LIN {X 0,Y 428.465,Z 323.366,A -85,B 0,C 180,E1 -10193.855,E2 -10193.855} C_VEL
LIN {X 0,Y 430.583,Z 198.986,A -85,B 0,C 180,E1 -10195.968,E2 -10195.968} C_VEL
LIN {X 0,Y 425.08,Z 170.607,A -85,B 0,C 180,E1 -10196.85,E2 -10196.85} C_VEL
LIN {X 0,Y 424.032,Z 165.531,A -85,B 0,C 180,E1 -10197.037,E2 -10197.037} C_VEL
LIN {X 0,Y 424.428,Z 159.339,A -85,B 0,C 180,E1 -10198.077,E2 -10198.077} C_VEL
LIN {X 0,Y 421.778,Z 147.828,A -85,B 0,C 180,E1 -10200.268,E2 -10200.268} C_VEL
LIN {X 0,Y 418.256,Z 134,A -85,B 0,C 180,E1 -10203.042,E2 -10203.042} C_VEL
LIN {X 0,Y 418.245,Z 134.011,A -85,B 0,C 180,E1 -10206.238,E2 -10206.238} C_VEL
LIN {X 0,Y 418.255,Z 134.011,A -85,B 0,C 180,E1 -10209.682,E2 -10209.682} C_VEL
LIN {X 0,Y 418.23,Z 134.011,A -85,B 0,C 180,E1 -10212.321,E2 -10212.321} C_VEL
LIN {X 0,Y 418.236,Z 134.01,A -85,B 0,C 180,E1 -10215.109,E2 -10215.109} C_VEL
LIN {X 0,Y 418.241,Z 134.014,A -85,B 0,C 180,E1 -10217.767,E2 -10217.767} C_VEL
LIN {X 0,Y 418.246,Z 134.008,A -85,B 0,C 180,E1 -10220.621,E2 -10220.621} C_VEL
LIN {X 0,Y 418.243,Z 134.006,A -85,B 0,C 180,E1 -10223.976,E2 -10223.976} C_VEL
LIN {X 0,Y 418.258,Z 134.007,A -85,B 0,C 180,E1 -10227.156,E2 -10227.156} C_VEL
LIN {X 0,Y 418.27,Z 134.005,A -85,B 0,C 180,E1 -10230.896,E2 -10230.896} C_VEL
LIN {X 0,Y 418.262,Z 134.006,A -85,B 0,C 180,E1 -10234.095,E2 -10234.095} C_VEL
LIN {X 0,Y 418.233,Z 134.014,A -85,B 0,C 180,E1 -10237.264,E2 -10237.264} C_VEL
LIN {X 0,Y 418.285,Z 134,A -85,B 0,C 180,E1 -10240.364,E2 -10240.364} C_VEL
LIN {X 0,Y 418.318,Z 133.997,A -85,B 0,C 180,E1 -10243.405,E2 -10243.405} C_VEL
LIN {X 0,Y 418.349,Z 133.994,A -85,B 0,C 180,E1 -10246.999,E2 -10246.999} C_VEL
LIN {X 0,Y 418.34,Z 134,A -85,B 0,C 180,E1 -10250.329,E2 -10250.329} C_VEL
LIN {X 0,Y 418.447,Z 133.985,A -85,B 0,C 180,E1 -10253.248,E2 -10253.248} C_VEL
LIN {X 0,Y 418.331,Z 133.995,A -85,B 0,C 180,E1 -10255.182,E2 -10255.182} C_VEL
LIN {X 0,Y 418.543,Z 133.974,A -85,B 0,C 180,E1 -10258.076,E2 -10258.076} C_VEL
LIN {X 0,Y 418.475,Z 133.98,A -85,B 0,C 180,E1 -10260.962,E2 -10260.962} C_VEL
LIN {X 0,Y 418.475,Z 133.981,A -85,B 0,C 180,E1 -10262.888,E2 -10262.888} C_VEL
LIN {X 0,Y 418.446,Z 133.983,A -85,B 0,C 180,E1 -10266.472,E2 -10266.472} C_VEL
LIN {X 0,Y 418.338,Z 133.994,A -85,B 0,C 180,E1 -10269.672,E2 -10269.672} C_VEL
LIN {X 0,Y 418.349,Z 133.99,A -85,B 0,C 180,E1 -10273.001,E2 -10273.001} C_VEL
LIN {X 0,Y 418.266,Z 134.002,A -85,B 0,C 180,E1 -10276.713,E2 -10276.713} C_VEL
LIN {X 0,Y 418.272,Z 134.01,A -85,B 0,C 180,E1 -10279.79,E2 -10279.79} C_VEL
LIN {X 0,Y 418.23,Z 134.011,A -85,B 0,C 180,E1 -10282.737,E2 -10282.737} C_VEL
LIN {X 0,Y 418.22,Z 133.997,A -85,B 0,C 180,E1 -10285.908,E2 -10285.908} C_VEL
LIN {X 0,Y 418.26,Z 134.007,A -85,B 0,C 180,E1 -10289.162,E2 -10289.162} C_VEL
LIN {X 0,Y 418.253,Z 134.009,A -85,B 0,C 180,E1 -10292.842,E2 -10292.842} C_VEL
LIN {X 0,Y 418.244,Z 134.008,A -85,B 0,C 180,E1 -10296.237,E2 -10296.237} C_VEL
LIN {X 0,Y 418.2,Z 134.014,A -85,B 0,C 180,E1 -10299.688,E2 -10299.688} C_VEL
LIN {X 0,Y 418.208,Z 134.01,A -85,B 0,C 180,E1 -10302.318,E2 -10302.318} C_VEL
LIN {X 0,Y 418.236,Z 134.013,A -85,B 0,C 180,E1 -10305.109,E2 -10305.109} C_VEL
LIN {X 0,Y 418.22,Z 134.014,A -85,B 0,C 180,E1 -10307.764,E2 -10307.764} C_VEL
LIN {X 0,Y 418.234,Z 134.008,A -85,B 0,C 180,E1 -10311.556,E2 -10311.556} C_VEL
LIN {X 0,Y 418.249,Z 134.011,A -85,B 0,C 180,E1 -10315.158,E2 -10315.158} C_VEL
LIN {X 0,Y 418.231,Z 134.012,A -85,B 0,C 180,E1 -10317.471,E2 -10317.471} C_VEL
LIN {X 0,Y 418.23,Z 134.052,A -85,B 0,C 180,E1 -10320.387,E2 -10320.387} C_VEL
LIN {X 0,Y 421.031,Z 145.484,A -85,B 0,C 180,E1 -10322.84,E2 -10322.84} C_VEL
LIN {X 0,Y 429.208,Z 164.619,A -85,B 0,C 180,E1 -10323.755,E2 -10323.755} C_VEL
LIN {X 0,Y 430.881,Z 171.966,A -85,B 0,C 180,E1 -10323.999,E2 -10323.999} C_VEL
LIN {X 0,Y 429.409,Z 263.169,A -85,B 0,C 180,E1 -10325.558,E2 -10325.558} C_VEL
LIN {X 0,Y 428.499,Z 309.991,A -85,B 0,C 180,E1 -10326.371,E2 -10326.371} C_VEL
LIN {X 0,Y 427.945,Z 325.824,A -85,B 0,C 180,E1 -10326.84,E2 -10326.84} C_VEL
LIN {X 0,Y 427.226,Z 340.105,A -85,B 0,C 180,E1 -10327.449,E2 -10327.449} C_VEL
LIN {X 0,Y 426.226,Z 353.97,A -85,B 0,C 180,E1 -10328.223,E2 -10328.223} C_VEL
LIN {X 0,Y 425.128,Z 367.554,A -85,B 0,C 180,E1 -10329.18,E2 -10329.18} C_VEL
LIN {X 0,Y 423.916,Z 380.046,A -85,B 0,C 180,E1 -10330.258,E2 -10330.258} C_VEL
LIN {X 0,Y 422.659,Z 392.692,A -85,B 0,C 180,E1 -10331.583,E2 -10331.583} C_VEL
LIN {X 0,Y 422.09,Z 397.98,A -85,B 0,C 180,E1 -10332.219,E2 -10332.219} C_VEL
LIN {X 0,Y 421.003,Z 402.312,A -85,B 0,C 180,E1 -10332.748,E2 -10332.748} C_VEL
LIN {X 0,Y 417.508,Z 409.152,A -85,B 0,C 180,E1 -10333.603,E2 -10333.603} C_VEL
LIN {X 0,Y 414.011,Z 415.635,A -85,B 0,C 180,E1 -10334.522,E2 -10334.522} C_VEL
LIN {X 0,Y 412.934,Z 419.28,A -85,B 0,C 180,E1 -10335.146,E2 -10335.146} C_VEL
LIN {X 0,Y 412.042,Z 427.938,A -85,B 0,C 180,E1 -10336.899,E2 -10336.899} C_VEL
LIN {X 0,Y 411.312,Z 435.184,A -85,B 0,C 180,E1 -10338.668,E2 -10338.668} C_VEL
LIN {X 0,Y 410.743,Z 441.74,A -85,B 0,C 180,E1 -10340.645,E2 -10340.645} C_VEL
LIN {X 0,Y 410.372,Z 446.865,A -85,B 0,C 180,E1 -10342.62,E2 -10342.62} C_VEL
LIN {X 0,Y 410.202,Z 449.817,A -85,B 0,C 180,E1 -10344.1,E2 -10344.1} C_VEL
LIN {X 0,Y 409.983,Z 452.712,A -85,B 0,C 180,E1 -10346.068,E2 -10346.068} C_VEL
LIN {X 0,Y 410.007,Z 454.45,A -85,B 0,C 180,E1 -10348.035,E2 -10348.035} C_VEL
LIN {X 0,Y 409.926,Z 455.061,A -85,B 0,C 180,E1 -10350,E2 -10350} C_VEL
LIN {X 0,Y 410.008,Z 454.499,A -85,B 0,C 180,E1 -10351.965,E2 -10351.965} C_VEL
LIN {X 0,Y 409.982,Z 452.825,A -85,B 0,C 180,E1 -10353.932,E2 -10353.932} C_VEL
LIN {X 0,Y 410.196,Z 449.992,A -85,B 0,C 180,E1 -10355.9,E2 -10355.9} C_VEL
LIN {X 0,Y 410.412,Z 445.938,A -85,B 0,C 180,E1 -10357.874,E2 -10357.874} C_VEL
LIN {X 0,Y 410.836,Z 440.56,A -85,B 0,C 180,E1 -10359.85,E2 -10359.85} C_VEL
LIN {X 0,Y 411.558,Z 433.702,A -85,B 0,C 180,E1 -10361.825,E2 -10361.825} C_VEL
LIN {X 0,Y 412.329,Z 425.145,A -85,B 0,C 180,E1 -10363.806,E2 -10363.806} C_VEL
LIN {X 0,Y 413.311,Z 416.043,A -85,B 0,C 180,E1 -10365.534,E2 -10365.534} C_VEL
LIN {X 0,Y 414.401,Z 406.762,A -85,B 0,C 180,E1 -10367.011,E2 -10367.011} C_VEL
LIN {X 0,Y 415.638,Z 395.779,A -85,B 0,C 180,E1 -10368.48,E2 -10368.48} C_VEL
LIN {X 0,Y 416.851,Z 383.672,A -85,B 0,C 180,E1 -10369.835,E2 -10369.835} C_VEL
LIN {X 0,Y 418.229,Z 370.41,A -85,B 0,C 180,E1 -10371.051,E2 -10371.051} C_VEL
LIN {X 0,Y 419.418,Z 357.406,A -85,B 0,C 180,E1 -10372.02,E2 -10372.02} C_VEL
LIN {X 0,Y 420.458,Z 344.114,A -85,B 0,C 180,E1 -10372.816,E2 -10372.816} C_VEL
LIN {X 0,Y 421.252,Z 329.188,A -85,B 0,C 180,E1 -10373.513,E2 -10373.513} C_VEL
LIN {X 0,Y 421.917,Z 313.686,A -85,B 0,C 180,E1 -10374.021,E2 -10374.021} C_VEL
LIN {X 0,Y 422.441,Z 293.788,A -85,B 0,C 180,E1 -10374.414,E2 -10374.414} C_VEL
LIN {X 0,Y 424.553,Z 173.198,A -85,B 0,C 180,E1 -10376.498,E2 -10376.498} C_VEL
LIN {X 0,Y 422.784,Z 166.169,A -85,B 0,C 180,E1 -10376.75,E2 -10376.75} C_VEL
LIN {X 0,Y 413.744,Z 145.287,A -85,B 0,C 180,E1 -10377.816,E2 -10377.816} C_VEL
LIN {X 0,Y 411.193,Z 134.892,A -85,B 0,C 180,E1 -10380.173,E2 -10380.173} C_VEL
LIN {X 0,Y 411.203,Z 134.893,A -85,B 0,C 180,E1 -10383.156,E2 -10383.156} C_VEL
LIN {X 0,Y 411.188,Z 134.888,A -85,B 0,C 180,E1 -10386.551,E2 -10386.551} C_VEL
LIN {X 0,Y 411.163,Z 134.888,A -85,B 0,C 180,E1 -10389.719,E2 -10389.719} C_VEL
LIN {X 0,Y 411.161,Z 134.898,A -85,B 0,C 180,E1 -10393.135,E2 -10393.135} C_VEL
LIN {X 0,Y 411.164,Z 134.892,A -85,B 0,C 180,E1 -10395.882,E2 -10395.882} C_VEL
LIN {X 0,Y 411.159,Z 134.893,A -85,B 0,C 180,E1 -10399.493,E2 -10399.493} C_VEL
LIN {X 0,Y 411.183,Z 134.881,A -85,B 0,C 180,E1 -10402.025,E2 -10402.025} C_VEL
LIN {X 0,Y 411.203,Z 134.889,A -85,B 0,C 180,E1 -10405.124,E2 -10405.124} C_VEL
LIN {X 0,Y 411.16,Z 134.881,A -85,B 0,C 180,E1 -10408.002,E2 -10408.002} C_VEL
LIN {X 0,Y 411.17,Z 134.89,A -85,B 0,C 180,E1 -10411.406,E2 -10411.406} C_VEL
LIN {X 0,Y 411.19,Z 134.889,A -85,B 0,C 180,E1 -10414.941,E2 -10414.941} C_VEL
LIN {X 0,Y 411.204,Z 134.884,A -85,B 0,C 180,E1 -10417.913,E2 -10417.913} C_VEL
LIN {X 0,Y 411.217,Z 134.882,A -85,B 0,C 180,E1 -10421.051,E2 -10421.051} C_VEL
LIN {X 0,Y 411.214,Z 134.89,A -85,B 0,C 180,E1 -10424.13,E2 -10424.13} C_VEL
LIN {X 0,Y 411.306,Z 134.87,A -85,B 0,C 180,E1 -10427.166,E2 -10427.166} C_VEL
LIN {X 0,Y 411.291,Z 134.872,A -85,B 0,C 180,E1 -10430.161,E2 -10430.161} C_VEL
LIN {X 0,Y 411.393,Z 134.863,A -85,B 0,C 180,E1 -10433.132,E2 -10433.132} C_VEL
LIN {X 0,Y 411.29,Z 134.872,A -85,B 0,C 180,E1 -10435.099,E2 -10435.099} C_VEL
LIN {X 0,Y 411.505,Z 134.851,A -85,B 0,C 180,E1 -10438.042,E2 -10438.042} C_VEL
LIN {X 0,Y 411.518,Z 134.844,A -85,B 0,C 180,E1 -10440,E2 -10440} C_VEL
LIN {X 0,Y 411.45,Z 134.857,A -85,B 0,C 180,E1 -10442.937,E2 -10442.937} C_VEL
LIN {X 0,Y 411.436,Z 134.86,A -85,B 0,C 180,E1 -10445.882,E2 -10445.882} C_VEL
LIN {X 0,Y 411.321,Z 134.871,A -85,B 0,C 180,E1 -10448.846,E2 -10448.846} C_VEL
LIN {X 0,Y 411.286,Z 134.878,A -85,B 0,C 180,E1 -10451.833,E2 -10451.833} C_VEL
LIN {X 0,Y 411.26,Z 134.879,A -85,B 0,C 180,E1 -10454.853,E2 -10454.853} C_VEL
LIN {X 0,Y 411.247,Z 134.876,A -85,B 0,C 180,E1 -10457.915,E2 -10457.915} C_VEL
LIN {X 0,Y 411.199,Z 134.891,A -85,B 0,C 180,E1 -10461.034,E2 -10461.034} C_VEL
LIN {X 0,Y 411.219,Z 134.886,A -85,B 0,C 180,E1 -10464.216,E2 -10464.216} C_VEL
LIN {X 0,Y 411.21,Z 134.887,A -85,B 0,C 180,E1 -10467.481,E2 -10467.481} C_VEL
LIN {X 0,Y 411.191,Z 134.892,A -85,B 0,C 180,E1 -10470.847,E2 -10470.847} C_VEL
LIN {X 0,Y 411.206,Z 134.884,A -85,B 0,C 180,E1 -10474.333,E2 -10474.333} C_VEL
LIN {X 0,Y 411.193,Z 134.887,A -85,B 0,C 180,E1 -10477.974,E2 -10477.974} C_VEL
LIN {X 0,Y 411.165,Z 134.892,A -85,B 0,C 180,E1 -10481.228,E2 -10481.228} C_VEL
LIN {X 0,Y 411.177,Z 134.892,A -85,B 0,C 180,E1 -10484.49,E2 -10484.49} C_VEL
LIN {X 0,Y 411.178,Z 134.892,A -85,B 0,C 180,E1 -10488.194,E2 -10488.194} C_VEL
LIN {X 0,Y 411.221,Z 134.883,A -85,B 0,C 180,E1 -10490.776,E2 -10490.776} C_VEL
LIN {X 0,Y 411.199,Z 134.89,A -85,B 0,C 180,E1 -10494.471,E2 -10494.471} C_VEL
LIN {X 0,Y 411.233,Z 135.051,A -85,B 0,C 180,E1 -10496.554,E2 -10496.554} C_VEL
LIN {X 0,Y 415.194,Z 150.404,A -85,B 0,C 180,E1 -10499.687,E2 -10499.687} C_VEL
LIN {X 0,Y 417.697,Z 161.831,A -85,B 0,C 180,E1 -10501.893,E2 -10501.893} C_VEL
LIN {X 0,Y 417.456,Z 165.689,A -85,B 0,C 180,E1 -10502.52,E2 -10502.52} C_VEL
LIN {X 0,Y 423.748,Z 197.159,A -85,B 0,C 180,E1 -10503.543,E2 -10503.543} C_VEL
LIN {X 0,Y 424.206,Z 201.035,A -85,B 0,C 180,E1 -10503.645,E2 -10503.645} C_VEL
LIN {X 0,Y 421.785,Z 331.248,A -85,B 0,C 180,E1 -10505.906,E2 -10505.906} C_VEL
LIN {X 0,Y 421.081,Z 346.776,A -85,B 0,C 180,E1 -10506.353,E2 -10506.353} C_VEL
LIN {X 0,Y 420.166,Z 360.483,A -85,B 0,C 180,E1 -10506.921,E2 -10506.921} C_VEL
LIN {X 0,Y 419.09,Z 374.745,A -85,B 0,C 180,E1 -10507.703,E2 -10507.703} C_VEL
LIN {X 0,Y 417.787,Z 388.648,A -85,B 0,C 180,E1 -10508.668,E2 -10508.668} C_VEL
LIN {X 0,Y 416.552,Z 401.392,A -85,B 0,C 180,E1 -10509.765,E2 -10509.765} C_VEL
LIN {X 0,Y 415.164,Z 414.281,A -85,B 0,C 180,E1 -10511.11,E2 -10511.11} C_VEL
LIN {X 0,Y 414.085,Z 425.08,A -85,B 0,C 180,E1 -10512.467,E2 -10512.467} C_VEL
LIN {X 0,Y 412.895,Z 435.07,A -85,B 0,C 180,E1 -10513.943,E2 -10513.943} C_VEL
LIN {X 0,Y 411.914,Z 444.849,A -85,B 0,C 180,E1 -10515.676,E2 -10515.676} C_VEL
LIN {X 0,Y 411.212,Z 453.014,A -85,B 0,C 180,E1 -10517.414,E2 -10517.414} C_VEL
LIN {X 0,Y 410.668,Z 459.765,A -85,B 0,C 180,E1 -10519.149,E2 -10519.149} C_VEL
LIN {X 0,Y 410.235,Z 466.002,A -85,B 0,C 180,E1 -10521.13,E2 -10521.13} C_VEL
LIN {X 0,Y 410.056,Z 470.829,A -85,B 0,C 180,E1 -10523.109,E2 -10523.109} C_VEL
LIN {X 0,Y 409.935,Z 474.365,A -85,B 0,C 180,E1 -10525.082,E2 -10525.082} C_VEL
LIN {X 0,Y 409.903,Z 476.692,A -85,B 0,C 180,E1 -10527.052,E2 -10527.052} C_VEL
LIN {X 0,Y 409.932,Z 477.864,A -85,B 0,C 180,E1 -10529.018,E2 -10529.018} C_VEL
LIN {X 0,Y 409.932,Z 477.862,A -85,B 0,C 180,E1 -10530.982,E2 -10530.982} C_VEL
LIN {X 0,Y 409.903,Z 476.684,A -85,B 0,C 180,E1 -10532.948,E2 -10532.948} C_VEL
LIN {X 0,Y 409.939,Z 474.353,A -85,B 0,C 180,E1 -10534.917,E2 -10534.917} C_VEL
LIN {X 0,Y 410.06,Z 470.819,A -85,B 0,C 180,E1 -10536.891,E2 -10536.891} C_VEL
LIN {X 0,Y 410.235,Z 465.989,A -85,B 0,C 180,E1 -10538.87,E2 -10538.87} C_VEL
LIN {X 0,Y 410.664,Z 459.74,A -85,B 0,C 180,E1 -10540.851,E2 -10540.851} C_VEL
LIN {X 0,Y 411.262,Z 451.893,A -85,B 0,C 180,E1 -10542.836,E2 -10542.836} C_VEL
LIN {X 0,Y 412.053,Z 443.553,A -85,B 0,C 180,E1 -10544.571,E2 -10544.571} C_VEL
LIN {X 0,Y 413.032,Z 433.506,A -85,B 0,C 180,E1 -10546.305,E2 -10546.305} C_VEL
LIN {X 0,Y 414.258,Z 423.24,A -85,B 0,C 180,E1 -10547.781,E2 -10547.781} C_VEL
LIN {X 0,Y 415.514,Z 411.006,A -85,B 0,C 180,E1 -10549.258,E2 -10549.258} C_VEL
LIN {X 0,Y 416.935,Z 397.391,A -85,B 0,C 180,E1 -10550.602,E2 -10550.602} C_VEL
LIN {X 0,Y 418.277,Z 383.744,A -85,B 0,C 180,E1 -10551.694,E2 -10551.694} C_VEL
LIN {X 0,Y 419.539,Z 369.612,A -85,B 0,C 180,E1 -10552.597,E2 -10552.597} C_VEL
LIN {X 0,Y 420.59,Z 354.722,A -85,B 0,C 180,E1 -10553.333,E2 -10553.333} C_VEL
LIN {X 0,Y 421.448,Z 339.122,A -85,B 0,C 180,E1 -10553.886,E2 -10553.886} C_VEL
LIN {X 0,Y 421.991,Z 323.148,A -85,B 0,C 180,E1 -10554.245,E2 -10554.245} C_VEL
LIN {X 0,Y 424.19,Z 200.35,A -85,B 0,C 180,E1 -10556.36,E2 -10556.36} C_VEL
LIN {X 0,Y 419.087,Z 173.276,A -85,B 0,C 180,E1 -10557.212,E2 -10557.212} C_VEL
LIN {X 0,Y 417.4,Z 165.401,A -85,B 0,C 180,E1 -10557.49,E2 -10557.49} C_VEL
LIN {X 0,Y 417.689,Z 161.765,A -85,B 0,C 180,E1 -10558.107,E2 -10558.107} C_VEL
LIN {X 0,Y 415.163,Z 150.385,A -85,B 0,C 180,E1 -10560.306,E2 -10560.306} C_VEL
LIN {X 0,Y 411.633,Z 136.549,A -85,B 0,C 180,E1 -10563.117,E2 -10563.117} C_VEL
LIN {X 0,Y 411.212,Z 134.879,A -85,B 0,C 180,E1 -10563.484,E2 -10563.484} C_VEL
LIN {X 0,Y 411.19,Z 134.89,A -85,B 0,C 180,E1 -10566.742,E2 -10566.742} C_VEL
LIN {X 0,Y 411.219,Z 134.888,A -85,B 0,C 180,E1 -10569.729,E2 -10569.729} C_VEL
LIN {X 0,Y 411.174,Z 134.89,A -85,B 0,C 180,E1 -10573.134,E2 -10573.134} C_VEL
LIN {X 0,Y 411.168,Z 134.894,A -85,B 0,C 180,E1 -10575.881,E2 -10575.881} C_VEL
LIN {X 0,Y 411.164,Z 134.891,A -85,B 0,C 180,E1 -10578.772,E2 -10578.772} C_VEL
LIN {X 0,Y 411.192,Z 134.887,A -85,B 0,C 180,E1 -10582.026,E2 -10582.026} C_VEL
LIN {X 0,Y 411.206,Z 134.887,A -85,B 0,C 180,E1 -10585.667,E2 -10585.667} C_VEL
LIN {X 0,Y 411.191,Z 134.89,A -85,B 0,C 180,E1 -10589.153,E2 -10589.153} C_VEL
LIN {X 0,Y 411.26,Z 134.879,A -85,B 0,C 180,E1 -10592.523,E2 -10592.523} C_VEL
LIN {X 0,Y 411.212,Z 134.883,A -85,B 0,C 180,E1 -10595.784,E2 -10595.784} C_VEL
LIN {X 0,Y 411.198,Z 134.89,A -85,B 0,C 180,E1 -10598.966,E2 -10598.966} C_VEL
LIN {X 0,Y 411.247,Z 134.881,A -85,B 0,C 180,E1 -10602.085,E2 -10602.085} C_VEL
LIN {X 0,Y 411.261,Z 134.882,A -85,B 0,C 180,E1 -10605.147,E2 -10605.147} C_VEL
LIN {X 0,Y 411.285,Z 134.872,A -85,B 0,C 180,E1 -10608.167,E2 -10608.167} C_VEL
LIN {X 0,Y 411.321,Z 134.867,A -85,B 0,C 180,E1 -10611.154,E2 -10611.154} C_VEL
LIN {X 0,Y 411.436,Z 134.859,A -85,B 0,C 180,E1 -10614.118,E2 -10614.118} C_VEL
LIN {X 0,Y 411.511,Z 134.85,A -85,B 0,C 180,E1 -10618.043,E2 -10618.043} C_VEL
LIN {X 0,Y 411.439,Z 134.856,A -85,B 0,C 180,E1 -10620.979,E2 -10620.979} C_VEL
LIN {X 0,Y 411.433,Z 134.858,A -85,B 0,C 180,E1 -10622.938,E2 -10622.938} C_VEL
LIN {X 0,Y 411.396,Z 134.861,A -85,B 0,C 180,E1 -10626.468,E2 -10626.468} C_VEL
LIN {X 0,Y 411.319,Z 134.867,A -85,B 0,C 180,E1 -10628.846,E2 -10628.846} C_VEL
LIN {X 0,Y 411.285,Z 134.88,A -85,B 0,C 180,E1 -10631.833,E2 -10631.833} C_VEL
LIN {X 0,Y 411.234,Z 134.883,A -85,B 0,C 180,E1 -10634.854,E2 -10634.854} C_VEL
LIN {X 0,Y 411.232,Z 134.883,A -85,B 0,C 180,E1 -10637.916,E2 -10637.916} C_VEL
LIN {X 0,Y 411.198,Z 134.883,A -85,B 0,C 180,E1 -10641.034,E2 -10641.034} C_VEL
LIN {X 0,Y 411.194,Z 134.884,A -85,B 0,C 180,E1 -10644.218,E2 -10644.218} C_VEL
LIN {X 0,Y 411.15,Z 134.88,A -85,B 0,C 180,E1 -10647.486,E2 -10647.486} C_VEL
LIN {X 0,Y 411.197,Z 134.892,A -85,B 0,C 180,E1 -10649.713,E2 -10649.713} C_VEL
LIN {X 0,Y 411.206,Z 134.889,A -85,B 0,C 180,E1 -10653.156,E2 -10653.156} C_VEL
LIN {X 0,Y 411.192,Z 134.887,A -85,B 0,C 180,E1 -10656.552,E2 -10656.552} C_VEL
LIN {X 0,Y 411.169,Z 134.889,A -85,B 0,C 180,E1 -10659.72,E2 -10659.72} C_VEL
LIN {X 0,Y 411.163,Z 134.893,A -85,B 0,C 180,E1 -10663.135,E2 -10663.135} C_VEL
LIN {X 0,Y 411.165,Z 134.892,A -85,B 0,C 180,E1 -10665.882,E2 -10665.882} C_VEL
LIN {X 0,Y 411.158,Z 134.896,A -85,B 0,C 180,E1 -10669.493,E2 -10669.493} C_VEL
LIN {X 0,Y 411.182,Z 134.888,A -85,B 0,C 180,E1 -10672.025,E2 -10672.025} C_VEL
LIN {X 0,Y 411.201,Z 134.888,A -85,B 0,C 180,E1 -10675.124,E2 -10675.124} C_VEL
LIN {X 0,Y 411.154,Z 134.896,A -85,B 0,C 180,E1 -10678.002,E2 -10678.002} C_VEL
LIN {X 0,Y 411.201,Z 134.938,A -85,B 0,C 180,E1 -10679.97,E2 -10679.97} C_VEL
LIN {X 0,Y 413.817,Z 145.548,A -85,B 0,C 180,E1 -10682.323,E2 -10682.323} C_VEL
LIN {X 0,Y 422.984,Z 166.753,A -85,B 0,C 180,E1 -10683.374,E2 -10683.374} C_VEL
LIN {X 0,Y 424.512,Z 173.264,A -85,B 0,C 180,E1 -10683.599,E2 -10683.599} C_VEL
LIN {X 0,Y 422.715,Z 275.901,A -85,B 0,C 180,E1 -10685.374,E2 -10685.374} C_VEL
LIN {X 0,Y 421.98,Z 311.398,A -85,B 0,C 180,E1 -10686.016,E2 -10686.016} C_VEL
LIN {X 0,Y 421.369,Z 326.831,A -85,B 0,C 180,E1 -10686.49,E2 -10686.49} C_VEL
LIN {X 0,Y 420.551,Z 342.01,A -85,B 0,C 180,E1 -10687.166,E2 -10687.166} C_VEL
LIN {X 0,Y 419.475,Z 356.065,A -85,B 0,C 180,E1 -10687.983,E2 -10687.983} C_VEL
LIN {X 0,Y 418.342,Z 369.32,A -85,B 0,C 180,E1 -10688.955,E2 -10688.955} C_VEL
LIN {X 0,Y 416.968,Z 382.79,A -85,B 0,C 180,E1 -10690.171,E2 -10690.171} C_VEL
LIN {X 0,Y 415.701,Z 395.002,A -85,B 0,C 180,E1 -10691.519,E2 -10691.519} C_VEL
LIN {X 0,Y 414.461,Z 406.125,A -85,B 0,C 180,E1 -10692.992,E2 -10692.992} C_VEL
LIN {X 0,Y 413.24,Z 416.927,A -85,B 0,C 180,E1 -10694.716,E2 -10694.716} C_VEL
LIN {X 0,Y 412.934,Z 419.28,A -85,B 0,C 180,E1 -10695.146,E2 -10695.146} C_VEL
LIN {X 0,Y 411.891,Z 422.819,A -85,B 0,C 180,E1 -10695.79,E2 -10695.79} C_VEL
LIN {X 0,Y 408.532,Z 428.303,A -85,B 0,C 180,E1 -10696.844,E2 -10696.844} C_VEL
LIN {X 0,Y 405.204,Z 433.371,A -85,B 0,C 180,E1 -10697.954,E2 -10697.954} C_VEL
LIN {X 0,Y 404.227,Z 436.141,A -85,B 0,C 180,E1 -10698.68,E2 -10698.68} C_VEL
LIN {X 0,Y 403.696,Z 441.942,A -85,B 0,C 180,E1 -10700.48,E2 -10700.48} C_VEL
LIN {X 0,Y 403.309,Z 447.066,A -85,B 0,C 180,E1 -10702.49,E2 -10702.49} C_VEL
LIN {X 0,Y 403.123,Z 450.017,A -85,B 0,C 180,E1 -10703.996,E2 -10703.996} C_VEL
LIN {X 0,Y 402.903,Z 452.911,A -85,B 0,C 180,E1 -10705.999,E2 -10705.999} C_VEL
LIN {X 0,Y 402.921,Z 454.649,A -85,B 0,C 180,E1 -10708.001,E2 -10708.001} C_VEL
LIN {X 0,Y 402.85,Z 455.259,A -85,B 0,C 180,E1 -10710,E2 -10710} C_VEL
LIN {X 0,Y 402.921,Z 454.697,A -85,B 0,C 180,E1 -10711.999,E2 -10711.999} C_VEL
LIN {X 0,Y 402.902,Z 453.023,A -85,B 0,C 180,E1 -10714.001,E2 -10714.001} C_VEL
LIN {X 0,Y 403.118,Z 450.19,A -85,B 0,C 180,E1 -10716.004,E2 -10716.004} C_VEL
LIN {X 0,Y 403.368,Z 446.136,A -85,B 0,C 180,E1 -10718.012,E2 -10718.012} C_VEL
LIN {X 0,Y 403.805,Z 440.758,A -85,B 0,C 180,E1 -10720.023,E2 -10720.023} C_VEL
LIN {X 0,Y 404.594,Z 433.899,A -85,B 0,C 180,E1 -10722.031,E2 -10722.031} C_VEL
LIN {X 0,Y 405.394,Z 425.343,A -85,B 0,C 180,E1 -10724.046,E2 -10724.046} C_VEL
LIN {X 0,Y 406.43,Z 416.24,A -85,B 0,C 180,E1 -10725.804,E2 -10725.804} C_VEL
LIN {X 0,Y 407.559,Z 406.959,A -85,B 0,C 180,E1 -10727.305,E2 -10727.305} C_VEL
LIN {X 0,Y 408.967,Z 395.188,A -85,B 0,C 180,E1 -10728.897,E2 -10728.897} C_VEL
LIN {X 0,Y 410.299,Z 382.689,A -85,B 0,C 180,E1 -10730.296,E2 -10730.296} C_VEL
LIN {X 0,Y 411.733,Z 369.152,A -85,B 0,C 180,E1 -10731.53,E2 -10731.53} C_VEL
LIN {X 0,Y 412.993,Z 355.835,A -85,B 0,C 180,E1 -10732.513,E2 -10732.513} C_VEL
LIN {X 0,Y 414.075,Z 341.493,A -85,B 0,C 180,E1 -10733.353,E2 -10733.353} C_VEL
LIN {X 0,Y 414.955,Z 326.502,A -85,B 0,C 180,E1 -10734.017,E2 -10734.017} C_VEL
LIN {X 0,Y 415.549,Z 311.591,A -85,B 0,C 180,E1 -10734.479,E2 -10734.479} C_VEL
LIN {X 0,Y 416.507,Z 267.153,A -85,B 0,C 180,E1 -10735.285,E2 -10735.285} C_VEL
LIN {X 0,Y 418.165,Z 174.26,A -85,B 0,C 180,E1 -10736.919,E2 -10736.919} C_VEL
LIN {X 0,Y 416.735,Z 168.78,A -85,B 0,C 180,E1 -10737.123,E2 -10737.123} C_VEL
LIN {X 0,Y 407.737,Z 148.297,A -85,B 0,C 180,E1 -10738.179,E2 -10738.179} C_VEL
LIN {X 0,Y 406.574,Z 145.519,A -85,B 0,C 180,E1 -10738.347,E2 -10738.347} C_VEL
LIN {X 0,Y 404.145,Z 135.77,A -85,B 0,C 180,E1 -10740.61,E2 -10740.61} C_VEL
LIN {X 0,Y 404.136,Z 135.768,A -85,B 0,C 180,E1 -10743.813,E2 -10743.813} C_VEL
LIN {X 0,Y 404.13,Z 135.768,A -85,B 0,C 180,E1 -10746.873,E2 -10746.873} C_VEL
LIN {X 0,Y 404.118,Z 135.766,A -85,B 0,C 180,E1 -10750.075,E2 -10750.075} C_VEL
LIN {X 0,Y 404.141,Z 135.771,A -85,B 0,C 180,E1 -10753.082,E2 -10753.082} C_VEL
LIN {X 0,Y 404.121,Z 135.769,A -85,B 0,C 180,E1 -10755.922,E2 -10755.922} C_VEL
LIN {X 0,Y 404.102,Z 135.765,A -85,B 0,C 180,E1 -10758.633,E2 -10758.633} C_VEL
LIN {X 0,Y 404.139,Z 135.76,A -85,B 0,C 180,E1 -10761.495,E2 -10761.495} C_VEL
LIN {X 0,Y 404.174,Z 135.766,A -85,B 0,C 180,E1 -10764.983,E2 -10764.983} C_VEL
LIN {X 0,Y 404.135,Z 135.752,A -85,B 0,C 180,E1 -10768.444,E2 -10768.444} C_VEL
LIN {X 0,Y 404.149,Z 135.766,A -85,B 0,C 180,E1 -10770.862,E2 -10770.862} C_VEL
LIN {X 0,Y 404.154,Z 135.767,A -85,B 0,C 180,E1 -10774.723,E2 -10774.723} C_VEL
LIN {X 0,Y 404.168,Z 135.759,A -85,B 0,C 180,E1 -10777.508,E2 -10777.508} C_VEL
LIN {X 0,Y 404.162,Z 135.762,A -85,B 0,C 180,E1 -10780.707,E2 -10780.707} C_VEL
LIN {X 0,Y 404.184,Z 135.763,A -85,B 0,C 180,E1 -10783.846,E2 -10783.846} C_VEL
LIN {X 0,Y 404.286,Z 135.745,A -85,B 0,C 180,E1 -10786.939,E2 -10786.939} C_VEL
LIN {X 0,Y 404.257,Z 135.749,A -85,B 0,C 180,E1 -10789.988,E2 -10789.988} C_VEL
LIN {X 0,Y 404.343,Z 135.741,A -85,B 0,C 180,E1 -10793.011,E2 -10793.011} C_VEL
LIN {X 0,Y 404.261,Z 135.747,A -85,B 0,C 180,E1 -10795.013,E2 -10795.013} C_VEL
LIN {X 0,Y 404.474,Z 135.727,A -85,B 0,C 180,E1 -10798.008,E2 -10798.008} C_VEL
LIN {X 0,Y 404.353,Z 135.736,A -85,B 0,C 180,E1 -10800.996,E2 -10800.996} C_VEL
LIN {X 0,Y 404.408,Z 135.734,A -85,B 0,C 180,E1 -10802.988,E2 -10802.988} C_VEL
LIN {X 0,Y 404.384,Z 135.737,A -85,B 0,C 180,E1 -10805.985,E2 -10805.985} C_VEL
LIN {X 0,Y 404.268,Z 135.749,A -85,B 0,C 180,E1 -10809.001,E2 -10809.001} C_VEL
LIN {X 0,Y 404.259,Z 135.752,A -85,B 0,C 180,E1 -10812.041,E2 -10812.041} C_VEL
LIN {X 0,Y 404.207,Z 135.76,A -85,B 0,C 180,E1 -10815.118,E2 -10815.118} C_VEL
LIN {X 0,Y 404.206,Z 135.753,A -85,B 0,C 180,E1 -10818.238,E2 -10818.238} C_VEL
LIN {X 0,Y 404.141,Z 135.766,A -85,B 0,C 180,E1 -10821.419,E2 -10821.419} C_VEL
LIN {X 0,Y 404.169,Z 135.768,A -85,B 0,C 180,E1 -10824.666,E2 -10824.666} C_VEL
LIN {X 0,Y 404.169,Z 135.763,A -85,B 0,C 180,E1 -10828.001,E2 -10828.001} C_VEL
LIN {X 0,Y 404.14,Z 135.767,A -85,B 0,C 180,E1 -10831.558,E2 -10831.558} C_VEL
LIN {X 0,Y 404.185,Z 135.764,A -85,B 0,C 180,E1 -10835.016,E2 -10835.016} C_VEL
LIN {X 0,Y 404.152,Z 135.767,A -85,B 0,C 180,E1 -10838.757,E2 -10838.757} C_VEL
LIN {X 0,Y 404.124,Z 135.769,A -85,B 0,C 180,E1 -10841.599,E2 -10841.599} C_VEL
LIN {X 0,Y 404.146,Z 135.767,A -85,B 0,C 180,E1 -10844.522,E2 -10844.522} C_VEL
LIN {X 0,Y 404.138,Z 135.766,A -85,B 0,C 180,E1 -10847.295,E2 -10847.295} C_VEL
LIN {X 0,Y 404.17,Z 135.753,A -85,B 0,C 180,E1 -10849.955,E2 -10849.955} C_VEL
LIN {X 0,Y 404.137,Z 135.768,A -85,B 0,C 180,E1 -10853.125,E2 -10853.125} C_VEL
LIN {X 0,Y 404.172,Z 135.82,A -85,B 0,C 180,E1 -10856.078,E2 -10856.078} C_VEL
LIN {X 0,Y 408.091,Z 150.977,A -85,B 0,C 180,E1 -10859.246,E2 -10859.246} C_VEL
LIN {X 0,Y 410.854,Z 163.174,A -85,B 0,C 180,E1 -10861.661,E2 -10861.661} C_VEL
LIN {X 0,Y 410.808,Z 165.45,A -85,B 0,C 180,E1 -10862.036,E2 -10862.036} C_VEL
LIN {X 0,Y 416.996,Z 196.146,A -85,B 0,C 180,E1 -10863.064,E2 -10863.064} C_VEL
LIN {X 0,Y 417.844,Z 201.404,A -85,B 0,C 180,E1 -10863.222,E2 -10863.222} C_VEL
LIN {X 0,Y 415.314,Z 331.066,A -85,B 0,C 180,E1 -10865.506,E2 -10865.506} C_VEL
LIN {X 0,Y 414.571,Z 346.587,A -85,B 0,C 180,E1 -10865.959,E2 -10865.959} C_VEL
LIN {X 0,Y 413.504,Z 362.118,A -85,B 0,C 180,E1 -10866.621,E2 -10866.621} C_VEL
LIN {X 0,Y 412.35,Z 376.542,A -85,B 0,C 180,E1 -10867.45,E2 -10867.45} C_VEL
LIN {X 0,Y 410.989,Z 390.038,A -85,B 0,C 180,E1 -10868.429,E2 -10868.429} C_VEL
LIN {X 0,Y 409.573,Z 403.785,A -85,B 0,C 180,E1 -10869.667,E2 -10869.667} C_VEL
LIN {X 0,Y 408.277,Z 415.158,A -85,B 0,C 180,E1 -10870.909,E2 -10870.909} C_VEL
LIN {X 0,Y 407.036,Z 426.673,A -85,B 0,C 180,E1 -10872.412,E2 -10872.412} C_VEL
LIN {X 0,Y 405.849,Z 436.365,A -85,B 0,C 180,E1 -10873.915,E2 -10873.915} C_VEL
LIN {X 0,Y 404.814,Z 445.889,A -85,B 0,C 180,E1 -10875.676,E2 -10875.676} C_VEL
LIN {X 0,Y 404.118,Z 453.831,A -85,B 0,C 180,E1 -10877.444,E2 -10877.444} C_VEL
LIN {X 0,Y 403.486,Z 461.245,A -85,B 0,C 180,E1 -10879.462,E2 -10879.462} C_VEL
LIN {X 0,Y 403.118,Z 467.13,A -85,B 0,C 180,E1 -10881.478,E2 -10881.478} C_VEL
LIN {X 0,Y 402.981,Z 470.63,A -85,B 0,C 180,E1 -10882.988,E2 -10882.988} C_VEL
LIN {X 0,Y 402.851,Z 474.167,A -85,B 0,C 180,E1 -10884.996,E2 -10884.996} C_VEL
LIN {X 0,Y 402.801,Z 476.493,A -85,B 0,C 180,E1 -10887,E2 -10887} C_VEL
LIN {X 0,Y 402.859,Z 477.666,A -85,B 0,C 180,E1 -10889,E2 -10889} C_VEL
LIN {X 0,Y 402.859,Z 477.664,A -85,B 0,C 180,E1 -10891,E2 -10891} C_VEL
LIN {X 0,Y 402.801,Z 476.485,A -85,B 0,C 180,E1 -10893,E2 -10893} C_VEL
LIN {X 0,Y 402.856,Z 474.153,A -85,B 0,C 180,E1 -10895.004,E2 -10895.004} C_VEL
LIN {X 0,Y 402.983,Z 470.618,A -85,B 0,C 180,E1 -10897.012,E2 -10897.012} C_VEL
LIN {X 0,Y 403.178,Z 465.788,A -85,B 0,C 180,E1 -10899.026,E2 -10899.026} C_VEL
LIN {X 0,Y 403.65,Z 459.539,A -85,B 0,C 180,E1 -10901.042,E2 -10901.042} C_VEL
LIN {X 0,Y 404.213,Z 451.689,A -85,B 0,C 180,E1 -10903.063,E2 -10903.063} C_VEL
LIN {X 0,Y 405.125,Z 443.35,A -85,B 0,C 180,E1 -10904.826,E2 -10904.826} C_VEL
LIN {X 0,Y 406.153,Z 433.303,A -85,B 0,C 180,E1 -10906.59,E2 -10906.59} C_VEL
LIN {X 0,Y 407.568,Z 421.957,A -85,B 0,C 180,E1 -10908.232,E2 -10908.232} C_VEL
LIN {X 0,Y 408.859,Z 409.649,A -85,B 0,C 180,E1 -10909.715,E2 -10909.715} C_VEL
LIN {X 0,Y 410.254,Z 397.187,A -85,B 0,C 180,E1 -10910.953,E2 -10910.953} C_VEL
LIN {X 0,Y 411.66,Z 383.54,A -85,B 0,C 180,E1 -10912.061,E2 -10912.061} C_VEL
LIN {X 0,Y 412.972,Z 369.406,A -85,B 0,C 180,E1 -10912.976,E2 -10912.976} C_VEL
LIN {X 0,Y 414.101,Z 353.792,A -85,B 0,C 180,E1 -10913.752,E2 -10913.752} C_VEL
LIN {X 0,Y 414.961,Z 338.91,A -85,B 0,C 180,E1 -10914.283,E2 -10914.283} C_VEL
LIN {X 0,Y 415.543,Z 322.93,A -85,B 0,C 180,E1 -10914.646,E2 -10914.646} C_VEL
LIN {X 0,Y 417.753,Z 200.697,A -85,B 0,C 180,E1 -10916.788,E2 -10916.788} C_VEL
LIN {X 0,Y 412.6,Z 174.015,A -85,B 0,C 180,E1 -10917.658,E2 -10917.658} C_VEL
LIN {X 0,Y 410.791,Z 165.162,A -85,B 0,C 180,E1 -10917.976,E2 -10917.976} C_VEL
LIN {X 0,Y 410.556,Z 161.542,A -85,B 0,C 180,E1 -10918.64,E2 -10918.64} C_VEL
LIN {X 0,Y 407.569,Z 148.96,A -85,B 0,C 180,E1 -10921.152,E2 -10921.152} C_VEL
LIN {X 0,Y 404.161,Z 135.763,A -85,B 0,C 180,E1 -10923.961,E2 -10923.961} C_VEL
LIN {X 0,Y 404.137,Z 135.768,A -85,B 0,C 180,E1 -10926.875,E2 -10926.875} C_VEL
LIN {X 0,Y 404.149,Z 135.769,A -85,B 0,C 180,E1 -10930.08,E2 -10930.08} C_VEL
LIN {X 0,Y 404.154,Z 135.764,A -85,B 0,C 180,E1 -10933.084,E2 -10933.084} C_VEL
LIN {X 0,Y 404.148,Z 135.767,A -85,B 0,C 180,E1 -10935.926,E2 -10935.926} C_VEL
LIN {X 0,Y 404.119,Z 135.768,A -85,B 0,C 180,E1 -10938.635,E2 -10938.635} C_VEL
LIN {X 0,Y 404.151,Z 135.764,A -85,B 0,C 180,E1 -10941.493,E2 -10941.493} C_VEL
LIN {X 0,Y 404.185,Z 135.758,A -85,B 0,C 180,E1 -10944.984,E2 -10944.984} C_VEL
LIN {X 0,Y 404.143,Z 135.765,A -85,B 0,C 180,E1 -10948.554,E2 -10948.554} C_VEL
LIN {X 0,Y 404.196,Z 135.758,A -85,B 0,C 180,E1 -10952.001,E2 -10952.001} C_VEL
LIN {X 0,Y 404.171,Z 135.764,A -85,B 0,C 180,E1 -10955.334,E2 -10955.334} C_VEL
LIN {X 0,Y 404.14,Z 135.769,A -85,B 0,C 180,E1 -10958.581,E2 -10958.581} C_VEL
LIN {X 0,Y 404.206,Z 135.758,A -85,B 0,C 180,E1 -10961.762,E2 -10961.762} C_VEL
LIN {X 0,Y 404.207,Z 135.761,A -85,B 0,C 180,E1 -10964.882,E2 -10964.882} C_VEL
LIN {X 0,Y 404.258,Z 135.746,A -85,B 0,C 180,E1 -10967.959,E2 -10967.959} C_VEL
LIN {X 0,Y 404.268,Z 135.747,A -85,B 0,C 180,E1 -10970.999,E2 -10970.999} C_VEL
LIN {X 0,Y 404.384,Z 135.737,A -85,B 0,C 180,E1 -10974.015,E2 -10974.015} C_VEL
LIN {X 0,Y 404.48,Z 135.725,A -85,B 0,C 180,E1 -10978.009,E2 -10978.009} C_VEL
LIN {X 0,Y 404.404,Z 135.733,A -85,B 0,C 180,E1 -10980.996,E2 -10980.996} C_VEL
LIN {X 0,Y 404.393,Z 135.734,A -85,B 0,C 180,E1 -10982.989,E2 -10982.989} C_VEL
LIN {X 0,Y 404.349,Z 135.738,A -85,B 0,C 180,E1 -10986.462,E2 -10986.462} C_VEL
LIN {X 0,Y 404.266,Z 135.745,A -85,B 0,C 180,E1 -10989.002,E2 -10989.002} C_VEL
LIN {X 0,Y 404.258,Z 135.753,A -85,B 0,C 180,E1 -10992.042,E2 -10992.042} C_VEL
LIN {X 0,Y 404.178,Z 135.762,A -85,B 0,C 180,E1 -10995.119,E2 -10995.119} C_VEL
LIN {X 0,Y 404.196,Z 135.762,A -85,B 0,C 180,E1 -10998.239,E2 -10998.239} C_VEL
LIN {X 0,Y 404.14,Z 135.764,A -85,B 0,C 180,E1 -11001.419,E2 -11001.419} C_VEL
LIN {X 0,Y 404.137,Z 135.761,A -85,B 0,C 180,E1 -11004.668,E2 -11004.668} C_VEL
LIN {X 0,Y 404.107,Z 135.766,A -85,B 0,C 180,E1 -11008.006,E2 -11008.006} C_VEL
LIN {X 0,Y 404.144,Z 135.765,A -85,B 0,C 180,E1 -11010.285,E2 -11010.285} C_VEL
LIN {X 0,Y 404.139,Z 135.764,A -85,B 0,C 180,E1 -11013.813,E2 -11013.813} C_VEL
LIN {X 0,Y 404.135,Z 135.767,A -85,B 0,C 180,E1 -11016.874,E2 -11016.874} C_VEL
LIN {X 0,Y 404.118,Z 135.766,A -85,B 0,C 180,E1 -11020.075,E2 -11020.075} C_VEL
LIN {X 0,Y 404.143,Z 135.767,A -85,B 0,C 180,E1 -11023.082,E2 -11023.082} C_VEL
LIN {X 0,Y 404.121,Z 135.769,A -85,B 0,C 180,E1 -11025.922,E2 -11025.922} C_VEL
LIN {X 0,Y 404.102,Z 135.774,A -85,B 0,C 180,E1 -11028.633,E2 -11028.633} C_VEL
LIN {X 0,Y 404.138,Z 135.763,A -85,B 0,C 180,E1 -11031.495,E2 -11031.495} C_VEL
LIN {X 0,Y 404.172,Z 135.762,A -85,B 0,C 180,E1 -11034.982,E2 -11034.982} C_VEL
LIN {X 0,Y 404.131,Z 135.769,A -85,B 0,C 180,E1 -11038.444,E2 -11038.444} C_VEL
LIN {X 0,Y 404.158,Z 135.833,A -85,B 0,C 180,E1 -11039.535,E2 -11039.535} C_VEL
LIN {X 0,Y 406.708,Z 145.934,A -85,B 0,C 180,E1 -11041.799,E2 -11041.799} C_VEL
LIN {X 0,Y 416.472,Z 168.152,A -85,B 0,C 180,E1 -11042.946,E2 -11042.946} C_VEL
LIN {X 0,Y 418.038,Z 173.803,A -85,B 0,C 180,E1 -11043.164,E2 -11043.164} C_VEL
LIN {X 0,Y 417.394,Z 220.796,A -85,B 0,C 180,E1 -11044.005,E2 -11044.005} C_VEL
LIN {X 0,Y 415.554,Z 310.427,A -85,B 0,C 180,E1 -11045.588,E2 -11045.588} C_VEL
LIN {X 0,Y 414.972,Z 325.685,A -85,B 0,C 180,E1 -11046.049,E2 -11046.049} C_VEL
LIN {X 0,Y 414.202,Z 339.996,A -85,B 0,C 180,E1 -11046.672,E2 -11046.672} C_VEL
LIN {X 0,Y 413.237,Z 352.402,A -85,B 0,C 180,E1 -11047.369,E2 -11047.369} C_VEL
LIN {X 0,Y 411.994,Z 366.388,A -85,B 0,C 180,E1 -11048.353,E2 -11048.353} C_VEL
LIN {X 0,Y 410.658,Z 379.169,A -85,B 0,C 180,E1 -11049.461,E2 -11049.461} C_VEL
LIN {X 0,Y 409.214,Z 392.145,A -85,B 0,C 180,E1 -11050.838,E2 -11050.838} C_VEL
LIN {X 0,Y 408.008,Z 402.79,A -85,B 0,C 180,E1 -11052.197,E2 -11052.197} C_VEL
LIN {X 0,Y 406.855,Z 412.727,A -85,B 0,C 180,E1 -11053.698,E2 -11053.698} C_VEL
LIN {X 0,Y 405.695,Z 422.431,A -85,B 0,C 180,E1 -11055.452,E2 -11055.452} C_VEL
LIN {X 0,Y 404.904,Z 430.511,A -85,B 0,C 180,E1 -11057.214,E2 -11057.214} C_VEL
LIN {X 0,Y 404.227,Z 436.141,A -85,B 0,C 180,E1 -11058.68,E2 -11058.68} C_VEL
LIN {X 0,Y 403.261,Z 438.776,A -85,B 0,C 180,E1 -11059.421,E2 -11059.421} C_VEL
LIN {X 0,Y 400.035,Z 442.722,A -85,B 0,C 180,E1 -11060.636,E2 -11060.636} C_VEL
LIN {X 0,Y 396.947,Z 446.194,A -85,B 0,C 180,E1 -11061.899,E2 -11061.899} C_VEL
LIN {X 0,Y 396.214,Z 447.986,A -85,B 0,C 180,E1 -11062.706,E2 -11062.706} C_VEL
LIN {X 0,Y 395.975,Z 451.81,A -85,B 0,C 180,E1 -11064.909,E2 -11064.909} C_VEL
LIN {X 0,Y 395.819,Z 454.12,A -85,B 0,C 180,E1 -11066.947,E2 -11066.947} C_VEL
LIN {X 0,Y 395.794,Z 455.299,A -85,B 0,C 180,E1 -11068.983,E2 -11068.983} C_VEL
LIN {X 0,Y 395.795,Z 455.315,A -85,B 0,C 180,E1 -11071.017,E2 -11071.017} C_VEL
LIN {X 0,Y 395.818,Z 454.2,A -85,B 0,C 180,E1 -11073.053,E2 -11073.053} C_VEL
LIN {X 0,Y 395.972,Z 451.952,A -85,B 0,C 180,E1 -11075.091,E2 -11075.091} C_VEL
LIN {X 0,Y 396.201,Z 448.518,A -85,B 0,C 180,E1 -11077.133,E2 -11077.133} C_VEL
LIN {X 0,Y 396.532,Z 443.819,A -85,B 0,C 180,E1 -11079.179,E2 -11079.179} C_VEL
LIN {X 0,Y 397.075,Z 437.727,A -85,B 0,C 180,E1 -11081.227,E2 -11081.227} C_VEL
LIN {X 0,Y 397.91,Z 431.099,A -85,B 0,C 180,E1 -11083.014,E2 -11083.014} C_VEL
LIN {X 0,Y 398.904,Z 421.865,A -85,B 0,C 180,E1 -11085.062,E2 -11085.062} C_VEL
LIN {X 0,Y 400.132,Z 412.001,A -85,B 0,C 180,E1 -11086.847,E2 -11086.847} C_VEL
LIN {X 0,Y 401.642,Z 400.317,A -85,B 0,C 180,E1 -11088.583,E2 -11088.583} C_VEL
LIN {X 0,Y 402.984,Z 388.737,A -85,B 0,C 180,E1 -11090.014,E2 -11090.014} C_VEL
LIN {X 0,Y 404.39,Z 376.46,A -85,B 0,C 180,E1 -11091.272,E2 -11091.272} C_VEL
LIN {X 0,Y 405.805,Z 363.039,A -85,B 0,C 180,E1 -11092.396,E2 -11092.396} C_VEL
LIN {X 0,Y 407.015,Z 349.129,A -85,B 0,C 180,E1 -11093.333,E2 -11093.333} C_VEL
LIN {X 0,Y 408.008,Z 334.761,A -85,B 0,C 180,E1 -11094.086,E2 -11094.086} C_VEL
LIN {X 0,Y 408.808,Z 319.492,A -85,B 0,C 180,E1 -11094.673,E2 -11094.673} C_VEL
LIN {X 0,Y 409.358,Z 304.592,A -85,B 0,C 180,E1 -11095.044,E2 -11095.044} C_VEL
LIN {X 0,Y 411.917,Z 176.444,A -85,B 0,C 180,E1 -11097.322,E2 -11097.322} C_VEL
LIN {X 0,Y 410.814,Z 171.59,A -85,B 0,C 180,E1 -11097.496,E2 -11097.496} C_VEL
LIN {X 0,Y 402.044,Z 151.702,A -85,B 0,C 180,E1 -11098.549,E2 -11098.549} C_VEL
LIN {X 0,Y 399.381,Z 145.714,A -85,B 0,C 180,E1 -11098.91,E2 -11098.91} C_VEL
LIN {X 0,Y 397.102,Z 136.648,A -85,B 0,C 180,E1 -11101.065,E2 -11101.065} C_VEL
LIN {X 0,Y 397.115,Z 136.644,A -85,B 0,C 180,E1 -11104.495,E2 -11104.495} C_VEL
LIN {X 0,Y 397.086,Z 136.65,A -85,B 0,C 180,E1 -11108.277,E2 -11108.277} C_VEL
LIN {X 0,Y 397.047,Z 136.652,A -85,B 0,C 180,E1 -11110.914,E2 -11110.914} C_VEL
LIN {X 0,Y 397.087,Z 136.646,A -85,B 0,C 180,E1 -11113.651,E2 -11113.651} C_VEL
LIN {X 0,Y 397.091,Z 136.642,A -85,B 0,C 180,E1 -11116.523,E2 -11116.523} C_VEL
LIN {X 0,Y 397.087,Z 136.648,A -85,B 0,C 180,E1 -11120.419,E2 -11120.419} C_VEL
LIN {X 0,Y 397.095,Z 136.632,A -85,B 0,C 180,E1 -11123.004,E2 -11123.004} C_VEL
LIN {X 0,Y 397.113,Z 136.639,A -85,B 0,C 180,E1 -11126.727,E2 -11126.727} C_VEL
LIN {X 0,Y 397.115,Z 136.633,A -85,B 0,C 180,E1 -11130.295,E2 -11130.295} C_VEL
LIN {X 0,Y 397.076,Z 136.644,A -85,B 0,C 180,E1 -11133.737,E2 -11133.737} C_VEL
LIN {X 0,Y 397.101,Z 136.64,A -85,B 0,C 180,E1 -11137.085,E2 -11137.085} C_VEL
LIN {X 0,Y 397.147,Z 136.639,A -85,B 0,C 180,E1 -11140.353,E2 -11140.353} C_VEL
LIN {X 0,Y 397.13,Z 136.639,A -85,B 0,C 180,E1 -11143.551,E2 -11143.551} C_VEL
LIN {X 0,Y 397.232,Z 136.624,A -85,B 0,C 180,E1 -11146.703,E2 -11146.703} C_VEL
LIN {X 0,Y 397.217,Z 136.628,A -85,B 0,C 180,E1 -11149.809,E2 -11149.809} C_VEL
LIN {X 0,Y 397.296,Z 136.619,A -85,B 0,C 180,E1 -11152.887,E2 -11152.887} C_VEL
LIN {X 0,Y 397.232,Z 136.622,A -85,B 0,C 180,E1 -11154.925,E2 -11154.925} C_VEL
LIN {X 0,Y 397.443,Z 136.603,A -85,B 0,C 180,E1 -11157.973,E2 -11157.973} C_VEL
LIN {X 0,Y 397.324,Z 136.611,A -85,B 0,C 180,E1 -11161.013,E2 -11161.013} C_VEL
LIN {X 0,Y 397.368,Z 136.612,A -85,B 0,C 180,E1 -11163.041,E2 -11163.041} C_VEL
LIN {X 0,Y 397.335,Z 136.615,A -85,B 0,C 180,E1 -11166.092,E2 -11166.092} C_VEL
LIN {X 0,Y 397.238,Z 136.624,A -85,B 0,C 180,E1 -11169.162,E2 -11169.162} C_VEL
LIN {X 0,Y 397.222,Z 136.629,A -85,B 0,C 180,E1 -11172.258,E2 -11172.258} C_VEL
LIN {X 0,Y 397.18,Z 136.64,A -85,B 0,C 180,E1 -11175.392,E2 -11175.392} C_VEL
LIN {X 0,Y 397.16,Z 136.632,A -85,B 0,C 180,E1 -11178.573,E2 -11178.573} C_VEL
LIN {X 0,Y 397.099,Z 136.641,A -85,B 0,C 180,E1 -11181.818,E2 -11181.818} C_VEL
LIN {X 0,Y 397.125,Z 136.642,A -85,B 0,C 180,E1 -11185.134,E2 -11185.134} C_VEL
LIN {X 0,Y 397.101,Z 136.647,A -85,B 0,C 180,E1 -11188.545,E2 -11188.545} C_VEL
LIN {X 0,Y 397.08,Z 136.647,A -85,B 0,C 180,E1 -11192.071,E2 -11192.071} C_VEL
LIN {X 0,Y 397.12,Z 136.641,A -85,B 0,C 180,E1 -11195.503,E2 -11195.503} C_VEL
LIN {X 0,Y 397.128,Z 136.641,A -85,B 0,C 180,E1 -11198.861,E2 -11198.861} C_VEL
LIN {X 0,Y 397.07,Z 136.648,A -85,B 0,C 180,E1 -11202.267,E2 -11202.267} C_VEL
LIN {X 0,Y 397.088,Z 136.645,A -85,B 0,C 180,E1 -11205.069,E2 -11205.069} C_VEL
LIN {X 0,Y 397.068,Z 136.651,A -85,B 0,C 180,E1 -11208.021,E2 -11208.021} C_VEL
LIN {X 0,Y 397.132,Z 136.639,A -85,B 0,C 180,E1 -11211.138,E2 -11211.138} C_VEL
LIN {X 0,Y 397.12,Z 136.643,A -85,B 0,C 180,E1 -11214.496,E2 -11214.496} C_VEL
LIN {X 0,Y 397.148,Z 136.728,A -85,B 0,C 180,E1 -11215.611,E2 -11215.611} C_VEL
LIN {X 0,Y 400.959,Z 151.53,A -85,B 0,C 180,E1 -11218.782,E2 -11218.782} C_VEL
LIN {X 0,Y 403.815,Z 163.608,A -85,B 0,C 180,E1 -11221.24,E2 -11221.24} C_VEL
LIN {X 0,Y 404.081,Z 165.137,A -85,B 0,C 180,E1 -11221.526,E2 -11221.526} C_VEL
LIN {X 0,Y 409.188,Z 189.319,A -85,B 0,C 180,E1 -11222.38,E2 -11222.38} C_VEL
LIN {X 0,Y 411.501,Z 202.086,A -85,B 0,C 180,E1 -11222.792,E2 -11222.792} C_VEL
LIN {X 0,Y 408.88,Z 330.884,A -85,B 0,C 180,E1 -11225.095,E2 -11225.095} C_VEL
LIN {X 0,Y 408.096,Z 346.398,A -85,B 0,C 180,E1 -11225.553,E2 -11225.553} C_VEL
LIN {X 0,Y 407.079,Z 360.656,A -85,B 0,C 180,E1 -11226.163,E2 -11226.163} C_VEL
LIN {X 0,Y 405.969,Z 374.358,A -85,B 0,C 180,E1 -11226.941,E2 -11226.941} C_VEL
LIN {X 0,Y 404.558,Z 388.258,A -85,B 0,C 180,E1 -11227.934,E2 -11227.934} C_VEL
LIN {X 0,Y 403.125,Z 400.997,A -85,B 0,C 180,E1 -11229.06,E2 -11229.06} C_VEL
LIN {X 0,Y 401.602,Z 413.885,A -85,B 0,C 180,E1 -11230.446,E2 -11230.446} C_VEL
LIN {X 0,Y 400.462,Z 424.684,A -85,B 0,C 180,E1 -11231.85,E2 -11231.85} C_VEL
LIN {X 0,Y 399.113,Z 434.671,A -85,B 0,C 180,E1 -11233.372,E2 -11233.372} C_VEL
LIN {X 0,Y 398.026,Z 444.451,A -85,B 0,C 180,E1 -11235.165,E2 -11235.165} C_VEL
LIN {X 0,Y 397.152,Z 452.338,A -85,B 0,C 180,E1 -11236.891,E2 -11236.891} C_VEL
LIN {X 0,Y 396.617,Z 459.367,A -85,B 0,C 180,E1 -11238.76,E2 -11238.76} C_VEL
LIN {X 0,Y 396.094,Z 465.603,A -85,B 0,C 180,E1 -11240.811,E2 -11240.811} C_VEL
LIN {X 0,Y 395.905,Z 470.431,A -85,B 0,C 180,E1 -11242.862,E2 -11242.862} C_VEL
LIN {X 0,Y 395.752,Z 473.968,A -85,B 0,C 180,E1 -11244.906,E2 -11244.906} C_VEL
LIN {X 0,Y 395.703,Z 476.295,A -85,B 0,C 180,E1 -11246.946,E2 -11246.946} C_VEL
LIN {X 0,Y 395.788,Z 477.468,A -85,B 0,C 180,E1 -11248.982,E2 -11248.982} C_VEL
LIN {X 0,Y 395.788,Z 477.466,A -85,B 0,C 180,E1 -11251.017,E2 -11251.017} C_VEL
LIN {X 0,Y 395.703,Z 476.285,A -85,B 0,C 180,E1 -11253.054,E2 -11253.054} C_VEL
LIN {X 0,Y 395.758,Z 473.953,A -85,B 0,C 180,E1 -11255.094,E2 -11255.094} C_VEL
LIN {X 0,Y 395.906,Z 470.418,A -85,B 0,C 180,E1 -11257.138,E2 -11257.138} C_VEL
LIN {X 0,Y 396.094,Z 465.587,A -85,B 0,C 180,E1 -11259.189,E2 -11259.189} C_VEL
LIN {X 0,Y 396.609,Z 459.337,A -85,B 0,C 180,E1 -11261.24,E2 -11261.24} C_VEL
LIN {X 0,Y 397.227,Z 451.384,A -85,B 0,C 180,E1 -11263.321,E2 -11263.321} C_VEL
LIN {X 0,Y 398.182,Z 443.147,A -85,B 0,C 180,E1 -11265.09,E2 -11265.09} C_VEL
LIN {X 0,Y 399.305,Z 433.101,A -85,B 0,C 180,E1 -11266.882,E2 -11266.882} C_VEL
LIN {X 0,Y 400.632,Z 422.834,A -85,B 0,C 180,E1 -11268.407,E2 -11268.407} C_VEL
LIN {X 0,Y 401.988,Z 410.598,A -85,B 0,C 180,E1 -11269.933,E2 -11269.933} C_VEL
LIN {X 0,Y 403.586,Z 396.983,A -85,B 0,C 180,E1 -11271.316,E2 -11271.316} C_VEL
LIN {X 0,Y 405.059,Z 383.335,A -85,B 0,C 180,E1 -11272.44,E2 -11272.44} C_VEL
LIN {X 0,Y 406.424,Z 369.201,A -85,B 0,C 180,E1 -11273.368,E2 -11273.368} C_VEL
LIN {X 0,Y 407.568,Z 354.018,A -85,B 0,C 180,E1 -11274.138,E2 -11274.138} C_VEL
LIN {X 0,Y 408.479,Z 338.698,A -85,B 0,C 180,E1 -11274.694,E2 -11274.694} C_VEL
LIN {X 0,Y 409.09,Z 322.711,A -85,B 0,C 180,E1 -11275.061,E2 -11275.061} C_VEL
LIN {X 0,Y 411.415,Z 201.669,A -85,B 0,C 180,E1 -11277.211,E2 -11277.211} C_VEL
LIN {X 0,Y 406.304,Z 175.256,A -85,B 0,C 180,E1 -11278.095,E2 -11278.095} C_VEL
LIN {X 0,Y 404.048,Z 164.936,A -85,B 0,C 180,E1 -11278.487,E2 -11278.487} C_VEL
LIN {X 0,Y 401.328,Z 152.999,A -85,B 0,C 180,E1 -11280.898,E2 -11280.898} C_VEL
LIN {X 0,Y 398.115,Z 140.344,A -85,B 0,C 180,E1 -11283.58,E2 -11283.58} C_VEL
LIN {X 0,Y 397.131,Z 136.638,A -85,B 0,C 180,E1 -11284.441,E2 -11284.441} C_VEL
LIN {X 0,Y 397.105,Z 136.647,A -85,B 0,C 180,E1 -11288.275,E2 -11288.275} C_VEL
LIN {X 0,Y 397.09,Z 136.644,A -85,B 0,C 180,E1 -11290.909,E2 -11290.909} C_VEL
LIN {X 0,Y 397.102,Z 136.648,A -85,B 0,C 180,E1 -11293.649,E2 -11293.649} C_VEL
LIN {X 0,Y 397.103,Z 136.641,A -85,B 0,C 180,E1 -11296.521,E2 -11296.521} C_VEL
LIN {X 0,Y 397.113,Z 136.641,A -85,B 0,C 180,E1 -11300.423,E2 -11300.423} C_VEL
LIN {X 0,Y 397.108,Z 136.637,A -85,B 0,C 180,E1 -11304.266,E2 -11304.266} C_VEL
LIN {X 0,Y 397.115,Z 136.639,A -85,B 0,C 180,E1 -11306.727,E2 -11306.727} C_VEL
LIN {X 0,Y 397.126,Z 136.635,A -85,B 0,C 180,E1 -11310.296,E2 -11310.296} C_VEL
LIN {X 0,Y 397.195,Z 136.631,A -85,B 0,C 180,E1 -11312.61,E2 -11312.61} C_VEL
LIN {X 0,Y 397.126,Z 136.637,A -85,B 0,C 180,E1 -11315.981,E2 -11315.981} C_VEL
LIN {X 0,Y 397.141,Z 136.633,A -85,B 0,C 180,E1 -11319.705,E2 -11319.705} C_VEL
LIN {X 0,Y 397.184,Z 136.634,A -85,B 0,C 180,E1 -11322.845,E2 -11322.845} C_VEL
LIN {X 0,Y 397.231,Z 136.628,A -85,B 0,C 180,E1 -11326.703,E2 -11326.703} C_VEL
LIN {X 0,Y 397.218,Z 136.629,A -85,B 0,C 180,E1 -11329.809,E2 -11329.809} C_VEL
LIN {X 0,Y 397.298,Z 136.622,A -85,B 0,C 180,E1 -11332.887,E2 -11332.887} C_VEL
LIN {X 0,Y 397.243,Z 136.623,A -85,B 0,C 180,E1 -11334.925,E2 -11334.925} C_VEL
LIN {X 0,Y 397.449,Z 136.601,A -85,B 0,C 180,E1 -11337.973,E2 -11337.973} C_VEL
LIN {X 0,Y 397.369,Z 136.609,A -85,B 0,C 180,E1 -11341.014,E2 -11341.014} C_VEL
LIN {X 0,Y 397.327,Z 136.614,A -85,B 0,C 180,E1 -11343.042,E2 -11343.042} C_VEL
LIN {X 0,Y 397.306,Z 136.617,A -85,B 0,C 180,E1 -11346.454,E2 -11346.454} C_VEL
LIN {X 0,Y 397.237,Z 136.62,A -85,B 0,C 180,E1 -11349.162,E2 -11349.162} C_VEL
LIN {X 0,Y 397.221,Z 136.626,A -85,B 0,C 180,E1 -11352.258,E2 -11352.258} C_VEL
LIN {X 0,Y 397.127,Z 136.641,A -85,B 0,C 180,E1 -11355.394,E2 -11355.394} C_VEL
LIN {X 0,Y 397.153,Z 136.637,A -85,B 0,C 180,E1 -11358.574,E2 -11358.574} C_VEL
LIN {X 0,Y 397.097,Z 136.644,A -85,B 0,C 180,E1 -11361.819,E2 -11361.819} C_VEL
LIN {X 0,Y 397.104,Z 136.636,A -85,B 0,C 180,E1 -11365.135,E2 -11365.135} C_VEL
LIN {X 0,Y 397.066,Z 136.645,A -85,B 0,C 180,E1 -11368.548,E2 -11368.548} C_VEL
LIN {X 0,Y 397.082,Z 136.648,A -85,B 0,C 180,E1 -11371.836,E2 -11371.836} C_VEL
LIN {X 0,Y 397.121,Z 136.636,A -85,B 0,C 180,E1 -11374.494,E2 -11374.494} C_VEL
LIN {X 0,Y 397.092,Z 136.643,A -85,B 0,C 180,E1 -11378.276,E2 -11378.276} C_VEL
LIN {X 0,Y 397.052,Z 136.645,A -85,B 0,C 180,E1 -11381.976,E2 -11381.976} C_VEL
LIN {X 0,Y 397.086,Z 136.646,A -85,B 0,C 180,E1 -11385.069,E2 -11385.069} C_VEL
LIN {X 0,Y 397.052,Z 136.651,A -85,B 0,C 180,E1 -11388.024,E2 -11388.024} C_VEL
LIN {X 0,Y 397.09,Z 136.641,A -85,B 0,C 180,E1 -11391.723,E2 -11391.723} C_VEL
LIN {X 0,Y 397.116,Z 136.645,A -85,B 0,C 180,E1 -11395.506,E2 -11395.506} C_VEL
LIN {X 0,Y 397.107,Z 136.735,A -85,B 0,C 180,E1 -11399.083,E2 -11399.083} C_VEL
LIN {X 0,Y 399.473,Z 146.027,A -85,B 0,C 180,E1 -11401.238,E2 -11401.238} C_VEL
LIN {X 0,Y 409.953,Z 169.563,A -85,B 0,C 180,E1 -11402.503,E2 -11402.503} C_VEL
LIN {X 0,Y 411.332,Z 173.607,A -85,B 0,C 180,E1 -11402.682,E2 -11402.682} C_VEL
LIN {X 0,Y 411.866,Z 176.652,A -85,B 0,C 180,E1 -11402.779,E2 -11402.779} C_VEL
LIN {X 0,Y 409.795,Z 278.137,A -85,B 0,C 180,E1 -11404.578,E2 -11404.578} C_VEL
LIN {X 0,Y 409.09,Z 311.827,A -85,B 0,C 180,E1 -11405.21,E2 -11405.21} C_VEL
LIN {X 0,Y 408.449,Z 326.771,A -85,B 0,C 180,E1 -11405.678,E2 -11405.678} C_VEL
LIN {X 0,Y 407.582,Z 341.734,A -85,B 0,C 180,E1 -11406.354,E2 -11406.354} C_VEL
LIN {X 0,Y 406.545,Z 354.587,A -85,B 0,C 180,E1 -11407.11,E2 -11407.11} C_VEL
LIN {X 0,Y 405.233,Z 368.17,A -85,B 0,C 180,E1 -11408.107,E2 -11408.107} C_VEL
LIN {X 0,Y 403.743,Z 381.944,A -85,B 0,C 180,E1 -11409.36,E2 -11409.36} C_VEL
LIN {X 0,Y 402.384,Z 393.304,A -85,B 0,C 180,E1 -11410.619,E2 -11410.619} C_VEL
LIN {X 0,Y 401.036,Z 404.763,A -85,B 0,C 180,E1 -11412.141,E2 -11412.141} C_VEL
LIN {X 0,Y 399.841,Z 414.405,A -85,B 0,C 180,E1 -11413.666,E2 -11413.666} C_VEL
LIN {X 0,Y 398.652,Z 423.854,A -85,B 0,C 180,E1 -11415.45,E2 -11415.45} C_VEL
LIN {X 0,Y 397.828,Z 431.714,A -85,B 0,C 180,E1 -11417.243,E2 -11417.243} C_VEL
LIN {X 0,Y 396.947,Z 439.054,A -85,B 0,C 180,E1 -11419.286,E2 -11419.286} C_VEL
LIN {X 0,Y 396.453,Z 444.874,A -85,B 0,C 180,E1 -11421.334,E2 -11421.334} C_VEL
LIN {X 0,Y 396.214,Z 447.986,A -85,B 0,C 180,E1 -11422.706,E2 -11422.706} C_VEL
LIN {X 0,Y 395.481,Z 449.628,A -85,B 0,C 180,E1 -11423.52,E2 -11423.52} C_VEL
LIN {X 0,Y 392.455,Z 451.936,A -85,B 0,C 180,E1 -11424.85,E2 -11424.85} C_VEL
LIN {X 0,Y 389.906,Z 453.397,A -85,B 0,C 180,E1 -11425.938,E2 -11425.938} C_VEL
LIN {X 0,Y 388.807,Z 454.238,A -85,B 0,C 180,E1 -11426.788,E2 -11426.788} C_VEL
LIN {X 0,Y 388.715,Z 454.45,A -85,B 0,C 180,E1 -11427.078,E2 -11427.078} C_VEL
LIN {X 0,Y 388.726,Z 455.497,A -85,B 0,C 180,E1 -11428.964,E2 -11428.964} C_VEL
LIN {X 0,Y 388.726,Z 455.513,A -85,B 0,C 180,E1 -11431.036,E2 -11431.036} C_VEL
LIN {X 0,Y 388.721,Z 454.398,A -85,B 0,C 180,E1 -11433.109,E2 -11433.109} C_VEL
LIN {X 0,Y 388.891,Z 452.15,A -85,B 0,C 180,E1 -11435.184,E2 -11435.184} C_VEL
LIN {X 0,Y 389.119,Z 448.717,A -85,B 0,C 180,E1 -11437.263,E2 -11437.263} C_VEL
LIN {X 0,Y 389.504,Z 444.017,A -85,B 0,C 180,E1 -11439.346,E2 -11439.346} C_VEL
LIN {X 0,Y 390.082,Z 437.925,A -85,B 0,C 180,E1 -11441.431,E2 -11441.431} C_VEL
LIN {X 0,Y 390.93,Z 431.298,A -85,B 0,C 180,E1 -11443.251,E2 -11443.251} C_VEL
LIN {X 0,Y 391.839,Z 423.294,A -85,B 0,C 180,E1 -11445.074,E2 -11445.074} C_VEL
LIN {X 0,Y 393.09,Z 413.683,A -85,B 0,C 180,E1 -11446.89,E2 -11446.89} C_VEL
LIN {X 0,Y 394.397,Z 403.854,A -85,B 0,C 180,E1 -11448.439,E2 -11448.439} C_VEL
LIN {X 0,Y 395.896,Z 392.16,A -85,B 0,C 180,E1 -11449.982,E2 -11449.982} C_VEL
LIN {X 0,Y 397.317,Z 380.518,A -85,B 0,C 180,E1 -11451.261,E2 -11451.261} C_VEL
LIN {X 0,Y 398.66,Z 367.966,A -85,B 0,C 180,E1 -11452.41,E2 -11452.41} C_VEL
LIN {X 0,Y 400.058,Z 354.278,A -85,B 0,C 180,E1 -11453.42,E2 -11453.42} C_VEL
LIN {X 0,Y 401.164,Z 340.588,A -85,B 0,C 180,E1 -11454.224,E2 -11454.224} C_VEL
LIN {X 0,Y 402.112,Z 325.158,A -85,B 0,C 180,E1 -11454.904,E2 -11454.904} C_VEL
LIN {X 0,Y 402.746,Z 310.76,A -85,B 0,C 180,E1 -11455.346,E2 -11455.346} C_VEL
LIN {X 0,Y 405.22,Z 196.004,A -85,B 0,C 180,E1 -11457.432,E2 -11457.432} C_VEL
LIN {X 0,Y 405.446,Z 176.24,A -85,B 0,C 180,E1 -11457.803,E2 -11457.803} C_VEL
LIN {X 0,Y 399.752,Z 162.418,A -85,B 0,C 180,E1 -11458.514,E2 -11458.514} C_VEL
LIN {X 0,Y 392.175,Z 145.94,A -85,B 0,C 180,E1 -11459.491,E2 -11459.491} C_VEL
LIN {X 0,Y 390.039,Z 137.528,A -85,B 0,C 180,E1 -11461.558,E2 -11461.558} C_VEL
LIN {X 0,Y 390.068,Z 137.528,A -85,B 0,C 180,E1 -11465.209,E2 -11465.209} C_VEL
LIN {X 0,Y 390.054,Z 137.52,A -85,B 0,C 180,E1 -11469.097,E2 -11469.097} C_VEL
LIN {X 0,Y 390.029,Z 137.526,A -85,B 0,C 180,E1 -11472.372,E2 -11472.372} C_VEL
LIN {X 0,Y 390.041,Z 137.526,A -85,B 0,C 180,E1 -11475.354,E2 -11475.354} C_VEL
LIN {X 0,Y 390.015,Z 137.516,A -85,B 0,C 180,E1 -11478.184,E2 -11478.184} C_VEL
LIN {X 0,Y 390.058,Z 137.519,A -85,B 0,C 180,E1 -11480.904,E2 -11480.904} C_VEL
LIN {X 0,Y 390.07,Z 137.521,A -85,B 0,C 180,E1 -11484.791,E2 -11484.791} C_VEL
LIN {X 0,Y 390.019,Z 137.508,A -85,B 0,C 180,E1 -11488.495,E2 -11488.495} C_VEL
LIN {X 0,Y 390.017,Z 137.527,A -85,B 0,C 180,E1 -11492.003,E2 -11492.003} C_VEL
LIN {X 0,Y 390.044,Z 137.522,A -85,B 0,C 180,E1 -11495.517,E2 -11495.517} C_VEL
LIN {X 0,Y 390.057,Z 137.521,A -85,B 0,C 180,E1 -11498.878,E2 -11498.878} C_VEL
LIN {X 0,Y 390.07,Z 137.517,A -85,B 0,C 180,E1 -11502.164,E2 -11502.164} C_VEL
LIN {X 0,Y 390.125,Z 137.511,A -85,B 0,C 180,E1 -11505.392,E2 -11505.392} C_VEL
LIN {X 0,Y 390.173,Z 137.504,A -85,B 0,C 180,E1 -11507.517,E2 -11507.517} C_VEL
LIN {X 0,Y 390.195,Z 137.496,A -85,B 0,C 180,E1 -11510.671,E2 -11510.671} C_VEL
LIN {X 0,Y 390.279,Z 137.495,A -85,B 0,C 180,E1 -11513.797,E2 -11513.797} C_VEL
LIN {X 0,Y 390.41,Z 137.479,A -85,B 0,C 180,E1 -11517.937,E2 -11517.937} C_VEL
LIN {X 0,Y 390.294,Z 137.487,A -85,B 0,C 180,E1 -11521.032,E2 -11521.032} C_VEL
LIN {X 0,Y 390.302,Z 137.492,A -85,B 0,C 180,E1 -11523.096,E2 -11523.096} C_VEL
LIN {X 0,Y 390.289,Z 137.492,A -85,B 0,C 180,E1 -11526.202,E2 -11526.202} C_VEL
LIN {X 0,Y 390.196,Z 137.501,A -85,B 0,C 180,E1 -11529.329,E2 -11529.329} C_VEL
LIN {X 0,Y 390.173,Z 137.507,A -85,B 0,C 180,E1 -11532.483,E2 -11532.483} C_VEL
LIN {X 0,Y 390.141,Z 137.514,A -85,B 0,C 180,E1 -11535.677,E2 -11535.677} C_VEL
LIN {X 0,Y 390.104,Z 137.513,A -85,B 0,C 180,E1 -11538.922,E2 -11538.922} C_VEL
LIN {X 0,Y 390.041,Z 137.52,A -85,B 0,C 180,E1 -11542.234,E2 -11542.234} C_VEL
LIN {X 0,Y 390.086,Z 137.515,A -85,B 0,C 180,E1 -11545.732,E2 -11545.732} C_VEL
LIN {X 0,Y 390.046,Z 137.525,A -85,B 0,C 180,E1 -11549.11,E2 -11549.11} C_VEL
LIN {X 0,Y 390.044,Z 137.523,A -85,B 0,C 180,E1 -11552.721,E2 -11552.721} C_VEL
LIN {X 0,Y 390.057,Z 137.521,A -85,B 0,C 180,E1 -11555.825,E2 -11555.825} C_VEL
LIN {X 0,Y 390.068,Z 137.518,A -85,B 0,C 180,E1 -11559.218,E2 -11559.218} C_VEL
LIN {X 0,Y 390.043,Z 137.523,A -85,B 0,C 180,E1 -11562.374,E2 -11562.374} C_VEL
LIN {X 0,Y 390.045,Z 137.522,A -85,B 0,C 180,E1 -11565.354,E2 -11565.354} C_VEL
LIN {X 0,Y 390.033,Z 137.526,A -85,B 0,C 180,E1 -11568.187,E2 -11568.187} C_VEL
LIN {X 0,Y 390.091,Z 137.515,A -85,B 0,C 180,E1 -11570.908,E2 -11570.908} C_VEL
LIN {X 0,Y 390.09,Z 137.518,A -85,B 0,C 180,E1 -11574.793,E2 -11574.793} C_VEL
LIN {X 0,Y 390.1,Z 137.647,A -85,B 0,C 180,E1 -11575.127,E2 -11575.127} C_VEL
LIN {X 0,Y 393.818,Z 151.749,A -85,B 0,C 180,E1 -11578.234,E2 -11578.234} C_VEL
LIN {X 0,Y 396.917,Z 164.989,A -85,B 0,C 180,E1 -11580.965,E2 -11580.965} C_VEL
LIN {X 0,Y 398.712,Z 170.118,A -85,B 0,C 180,E1 -11581.21,E2 -11581.21} C_VEL
LIN {X 0,Y 404.55,Z 199.594,A -85,B 0,C 180,E1 -11582.24,E2 -11582.24} C_VEL
LIN {X 0,Y 405.122,Z 203.893,A -85,B 0,C 180,E1 -11582.366,E2 -11582.366} C_VEL
LIN {X 0,Y 402.582,Z 326.185,A -85,B 0,C 180,E1 -11584.574,E2 -11584.574} C_VEL
LIN {X 0,Y 401.936,Z 341.63,A -85,B 0,C 180,E1 -11584.98,E2 -11584.98} C_VEL
LIN {X 0,Y 400.928,Z 355.851,A -85,B 0,C 180,E1 -11585.53,E2 -11585.53} C_VEL
LIN {X 0,Y 399.81,Z 370.179,A -85,B 0,C 180,E1 -11586.29,E2 -11586.29} C_VEL
LIN {X 0,Y 398.5,Z 383.272,A -85,B 0,C 180,E1 -11587.17,E2 -11587.17} C_VEL
LIN {X 0,Y 396.975,Z 396.88,A -85,B 0,C 180,E1 -11588.311,E2 -11588.311} C_VEL
LIN {X 0,Y 395.28,Z 410.465,A -85,B 0,C 180,E1 -11589.714,E2 -11589.714} C_VEL
LIN {X 0,Y 393.85,Z 422.693,A -85,B 0,C 180,E1 -11591.264,E2 -11591.264} C_VEL
LIN {X 0,Y 392.479,Z 432.955,A -85,B 0,C 180,E1 -11592.815,E2 -11592.815} C_VEL
LIN {X 0,Y 391.261,Z 442.991,A -85,B 0,C 180,E1 -11594.636,E2 -11594.636} C_VEL
LIN {X 0,Y 390.216,Z 451.706,A -85,B 0,C 180,E1 -11596.549,E2 -11596.549} C_VEL
LIN {X 0,Y 389.588,Z 459.167,A -85,B 0,C 180,E1 -11598.554,E2 -11598.554} C_VEL
LIN {X 0,Y 389.026,Z 465.403,A -85,B 0,C 180,E1 -11600.643,E2 -11600.643} C_VEL
LIN {X 0,Y 388.824,Z 470.232,A -85,B 0,C 180,E1 -11602.731,E2 -11602.731} C_VEL
LIN {X 0,Y 388.659,Z 473.769,A -85,B 0,C 180,E1 -11604.813,E2 -11604.813} C_VEL
LIN {X 0,Y 388.61,Z 476.096,A -85,B 0,C 180,E1 -11606.89,E2 -11606.89} C_VEL
LIN {X 0,Y 388.7,Z 477.269,A -85,B 0,C 180,E1 -11608.964,E2 -11608.964} C_VEL
LIN {X 0,Y 388.7,Z 477.267,A -85,B 0,C 180,E1 -11611.036,E2 -11611.036} C_VEL
LIN {X 0,Y 388.61,Z 476.086,A -85,B 0,C 180,E1 -11613.11,E2 -11613.11} C_VEL
LIN {X 0,Y 388.665,Z 473.754,A -85,B 0,C 180,E1 -11615.187,E2 -11615.187} C_VEL
LIN {X 0,Y 388.825,Z 470.217,A -85,B 0,C 180,E1 -11617.269,E2 -11617.269} C_VEL
LIN {X 0,Y 389.026,Z 465.385,A -85,B 0,C 180,E1 -11619.357,E2 -11619.357} C_VEL
LIN {X 0,Y 389.58,Z 459.135,A -85,B 0,C 180,E1 -11621.446,E2 -11621.446} C_VEL
LIN {X 0,Y 390.244,Z 451.284,A -85,B 0,C 180,E1 -11623.54,E2 -11623.54} C_VEL
LIN {X 0,Y 391.26,Z 442.945,A -85,B 0,C 180,E1 -11625.364,E2 -11625.364} C_VEL
LIN {X 0,Y 392.441,Z 432.898,A -85,B 0,C 180,E1 -11627.187,E2 -11627.187} C_VEL
LIN {X 0,Y 393.862,Z 422.103,A -85,B 0,C 180,E1 -11628.812,E2 -11628.812} C_VEL
LIN {X 0,Y 395.275,Z 410.395,A -85,B 0,C 180,E1 -11630.286,E2 -11630.286} C_VEL
LIN {X 0,Y 396.938,Z 396.779,A -85,B 0,C 180,E1 -11631.691,E2 -11631.691} C_VEL
LIN {X 0,Y 398.482,Z 383.131,A -85,B 0,C 180,E1 -11632.831,E2 -11632.831} C_VEL
LIN {X 0,Y 399.911,Z 368.996,A -85,B 0,C 180,E1 -11633.772,E2 -11633.772} C_VEL
LIN {X 0,Y 401.097,Z 353.501,A -85,B 0,C 180,E1 -11634.567,E2 -11634.567} C_VEL
LIN {X 0,Y 402.03,Z 338.487,A -85,B 0,C 180,E1 -11635.117,E2 -11635.117} C_VEL
LIN {X 0,Y 402.66,Z 322.492,A -85,B 0,C 180,E1 -11635.49,E2 -11635.49} C_VEL
LIN {X 0,Y 405.111,Z 202.804,A -85,B 0,C 180,E1 -11637.644,E2 -11637.644} C_VEL
LIN {X 0,Y 400.136,Z 177.083,A -85,B 0,C 180,E1 -11638.527,E2 -11638.527} C_VEL
LIN {X 0,Y 397.947,Z 167.588,A -85,B 0,C 180,E1 -11638.888,E2 -11638.888} C_VEL
LIN {X 0,Y 396.835,Z 164.67,A -85,B 0,C 180,E1 -11639.061,E2 -11639.061} C_VEL
LIN {X 0,Y 393.812,Z 151.668,A -85,B 0,C 180,E1 -11641.766,E2 -11641.766} C_VEL
LIN {X 0,Y 390.075,Z 137.517,A -85,B 0,C 180,E1 -11644.912,E2 -11644.912} C_VEL
LIN {X 0,Y 390.044,Z 137.524,A -85,B 0,C 180,E1 -11647.78,E2 -11647.78} C_VEL
LIN {X 0,Y 390.057,Z 137.52,A -85,B 0,C 180,E1 -11650.822,E2 -11650.822} C_VEL
LIN {X 0,Y 390.055,Z 137.524,A -85,B 0,C 180,E1 -11653.886,E2 -11653.886} C_VEL
LIN {X 0,Y 390.058,Z 137.519,A -85,B 0,C 180,E1 -11656.79,E2 -11656.79} C_VEL
LIN {X 0,Y 390.057,Z 137.521,A -85,B 0,C 180,E1 -11659.561,E2 -11659.561} C_VEL
LIN {X 0,Y 390.043,Z 137.521,A -85,B 0,C 180,E1 -11662.45,E2 -11662.45} C_VEL
LIN {X 0,Y 390.069,Z 137.517,A -85,B 0,C 180,E1 -11665.976,E2 -11665.976} C_VEL
LIN {X 0,Y 390.048,Z 137.518,A -85,B 0,C 180,E1 -11669.869,E2 -11669.869} C_VEL
LIN {X 0,Y 390.113,Z 137.513,A -85,B 0,C 180,E1 -11673.232,E2 -11673.232} C_VEL
LIN {X 0,Y 390.069,Z 137.518,A -85,B 0,C 180,E1 -11676.764,E2 -11676.764} C_VEL
LIN {X 0,Y 390.105,Z 137.509,A -85,B 0,C 180,E1 -11679.983,E2 -11679.983} C_VEL
LIN {X 0,Y 390.14,Z 137.507,A -85,B 0,C 180,E1 -11683.248,E2 -11683.248} C_VEL
LIN {X 0,Y 390.197,Z 137.506,A -85,B 0,C 180,E1 -11686.562,E2 -11686.562} C_VEL
LIN {X 0,Y 390.169,Z 137.507,A -85,B 0,C 180,E1 -11689.623,E2 -11689.623} C_VEL
LIN {X 0,Y 390.25,Z 137.498,A -85,B 0,C 180,E1 -11692.758,E2 -11692.758} C_VEL
LIN {X 0,Y 390.213,Z 137.5,A -85,B 0,C 180,E1 -11694.833,E2 -11694.833} C_VEL
LIN {X 0,Y 390.418,Z 137.477,A -85,B 0,C 180,E1 -11697.937,E2 -11697.937} C_VEL
LIN {X 0,Y 390.336,Z 137.485,A -85,B 0,C 180,E1 -11701.032,E2 -11701.032} C_VEL
LIN {X 0,Y 390.264,Z 137.494,A -85,B 0,C 180,E1 -11703.097,E2 -11703.097} C_VEL
LIN {X 0,Y 390.267,Z 137.495,A -85,B 0,C 180,E1 -11706.444,E2 -11706.444} C_VEL
LIN {X 0,Y 390.194,Z 137.498,A -85,B 0,C 180,E1 -11709.329,E2 -11709.329} C_VEL
LIN {X 0,Y 390.173,Z 137.502,A -85,B 0,C 180,E1 -11712.483,E2 -11712.483} C_VEL
LIN {X 0,Y 390.07,Z 137.523,A -85,B 0,C 180,E1 -11715.68,E2 -11715.68} C_VEL
LIN {X 0,Y 390.1,Z 137.515,A -85,B 0,C 180,E1 -11718.922,E2 -11718.922} C_VEL
LIN {X 0,Y 390.037,Z 137.525,A -85,B 0,C 180,E1 -11722.234,E2 -11722.234} C_VEL
LIN {X 0,Y 390.051,Z 137.505,A -85,B 0,C 180,E1 -11725.722,E2 -11725.722} C_VEL
LIN {X 0,Y 390.027,Z 137.524,A -85,B 0,C 180,E1 -11729.112,E2 -11729.112} C_VEL
LIN {X 0,Y 390.043,Z 137.523,A -85,B 0,C 180,E1 -11732.722,E2 -11732.722} C_VEL
LIN {X 0,Y 390.054,Z 137.522,A -85,B 0,C 180,E1 -11735.825,E2 -11735.825} C_VEL
LIN {X 0,Y 390.037,Z 137.524,A -85,B 0,C 180,E1 -11739.212,E2 -11739.212} C_VEL
LIN {X 0,Y 390.031,Z 137.52,A -85,B 0,C 180,E1 -11742.372,E2 -11742.372} C_VEL
LIN {X 0,Y 390.041,Z 137.526,A -85,B 0,C 180,E1 -11745.354,E2 -11745.354} C_VEL
LIN {X 0,Y 390.015,Z 137.528,A -85,B 0,C 180,E1 -11748.184,E2 -11748.184} C_VEL
LIN {X 0,Y 390.057,Z 137.518,A -85,B 0,C 180,E1 -11750.904,E2 -11750.904} C_VEL
LIN {X 0,Y 390.068,Z 137.517,A -85,B 0,C 180,E1 -11754.791,E2 -11754.791} C_VEL
LIN {X 0,Y 390.067,Z 137.63,A -85,B 0,C 180,E1 -11758.613,E2 -11758.613} C_VEL
LIN {X 0,Y 392.262,Z 146.21,A -85,B 0,C 180,E1 -11760.656,E2 -11760.656} C_VEL
LIN {X 0,Y 401.864,Z 167.238,A -85,B 0,C 180,E1 -11761.849,E2 -11761.849} C_VEL
LIN {X 0,Y 405.311,Z 176.081,A -85,B 0,C 180,E1 -11762.286,E2 -11762.286} C_VEL
LIN {X 0,Y 405.49,Z 180.565,A -85,B 0,C 180,E1 -11762.387,E2 -11762.387} C_VEL
LIN {X 0,Y 403.489,Z 276.573,A -85,B 0,C 180,E1 -11764.117,E2 -11764.117} C_VEL
LIN {X 0,Y 402.678,Z 312.042,A -85,B 0,C 180,E1 -11764.788,E2 -11764.788} C_VEL
LIN {X 0,Y 402.068,Z 326.227,A -85,B 0,C 180,E1 -11765.234,E2 -11765.234} C_VEL
LIN {X 0,Y 401.157,Z 341.269,A -85,B 0,C 180,E1 -11765.913,E2 -11765.913} C_VEL
LIN {X 0,Y 400.011,Z 354.793,A -85,B 0,C 180,E1 -11766.714,E2 -11766.714} C_VEL
LIN {X 0,Y 398.64,Z 368.374,A -85,B 0,C 180,E1 -11767.725,E2 -11767.725} C_VEL
LIN {X 0,Y 397.078,Z 382.149,A -85,B 0,C 180,E1 -11768.997,E2 -11768.997} C_VEL
LIN {X 0,Y 395.555,Z 394.608,A -85,B 0,C 180,E1 -11770.41,E2 -11770.41} C_VEL
LIN {X 0,Y 394.248,Z 404.966,A -85,B 0,C 180,E1 -11771.822,E2 -11771.822} C_VEL
LIN {X 0,Y 393.001,Z 414.607,A -85,B 0,C 180,E1 -11773.374,E2 -11773.374} C_VEL
LIN {X 0,Y 391.737,Z 424.056,A -85,B 0,C 180,E1 -11775.188,E2 -11775.188} C_VEL
LIN {X 0,Y 390.869,Z 431.915,A -85,B 0,C 180,E1 -11777.011,E2 -11777.011} C_VEL
LIN {X 0,Y 389.936,Z 439.255,A -85,B 0,C 180,E1 -11779.091,E2 -11779.091} C_VEL
LIN {X 0,Y 389.399,Z 445.075,A -85,B 0,C 180,E1 -11781.175,E2 -11781.175} C_VEL
LIN {X 0,Y 389.126,Z 448.519,A -85,B 0,C 180,E1 -11782.737,E2 -11782.737} C_VEL
LIN {X 0,Y 388.893,Z 452.009,A -85,B 0,C 180,E1 -11784.816,E2 -11784.816} C_VEL
LIN {X 0,Y 388.715,Z 454.45,A -85,B 0,C 180,E1 -11787.078,E2 -11787.078} C_VEL
LIN {X 0,Y 388.035,Z 455.074,A -85,B 0,C 180,E1 -11787.94,E2 -11787.94} C_VEL
LIN {X 0,Y 385.159,Z 455.656,A -85,B 0,C 180,E1 -11789.344,E2 -11789.344} C_VEL
LIN {X 0,Y 382.736,Z 455.766,A -85,B 0,C 180,E1 -11790.481,E2 -11790.481} C_VEL
LIN {X 0,Y 381.704,Z 455.627,A -85,B 0,C 180,E1 -11791.359,E2 -11791.359} C_VEL
LIN {X 0,Y 381.624,Z 455.473,A -85,B 0,C 180,E1 -11791.656,E2 -11791.656} C_VEL
LIN {X 0,Y 381.627,Z 454.597,A -85,B 0,C 180,E1 -11793.167,E2 -11793.167} C_VEL
LIN {X 0,Y 381.814,Z 452.348,A -85,B 0,C 180,E1 -11795.281,E2 -11795.281} C_VEL
LIN {X 0,Y 382.051,Z 448.916,A -85,B 0,C 180,E1 -11797.398,E2 -11797.398} C_VEL
LIN {X 0,Y 382.456,Z 444.215,A -85,B 0,C 180,E1 -11799.52,E2 -11799.52} C_VEL
LIN {X 0,Y 383.1,Z 438.123,A -85,B 0,C 180,E1 -11801.642,E2 -11801.642} C_VEL
LIN {X 0,Y 383.966,Z 431.497,A -85,B 0,C 180,E1 -11803.496,E2 -11803.496} C_VEL
LIN {X 0,Y 385.12,Z 422.261,A -85,B 0,C 180,E1 -11805.615,E2 -11805.615} C_VEL
LIN {X 0,Y 386.527,Z 412.394,A -85,B 0,C 180,E1 -11807.458,E2 -11807.458} C_VEL
LIN {X 0,Y 388.15,Z 400.971,A -85,B 0,C 180,E1 -11809.216,E2 -11809.216} C_VEL
LIN {X 0,Y 389.597,Z 389.125,A -85,B 0,C 180,E1 -11810.733,E2 -11810.733} C_VEL
LIN {X 0,Y 391.161,Z 376.848,A -85,B 0,C 180,E1 -11812.028,E2 -11812.028} C_VEL
LIN {X 0,Y 392.515,Z 365.005,A -85,B 0,C 180,E1 -11813.059,E2 -11813.059} C_VEL
LIN {X 0,Y 393.746,Z 352.487,A -85,B 0,C 180,E1 -11813.958,E2 -11813.958} C_VEL
LIN {X 0,Y 394.896,Z 337.678,A -85,B 0,C 180,E1 -11814.802,E2 -11814.802} C_VEL
LIN {X 0,Y 395.819,Z 322.603,A -85,B 0,C 180,E1 -11815.434,E2 -11815.434} C_VEL
LIN {X 0,Y 396.459,Z 307.952,A -85,B 0,C 180,E1 -11815.847,E2 -11815.847} C_VEL
LIN {X 0,Y 399.261,Z 181.952,A -85,B 0,C 180,E1 -11818.161,E2 -11818.161} C_VEL
LIN {X 0,Y 399.172,Z 177.77,A -85,B 0,C 180,E1 -11818.252,E2 -11818.252} C_VEL
LIN {X 0,Y 389.988,Z 156.683,A -85,B 0,C 180,E1 -11819.421,E2 -11819.421} C_VEL
LIN {X 0,Y 385.036,Z 146.168,A -85,B 0,C 180,E1 -11820.092,E2 -11820.092} C_VEL
LIN {X 0,Y 383.005,Z 138.405,A -85,B 0,C 180,E1 -11822.034,E2 -11822.034} C_VEL
LIN {X 0,Y 383.011,Z 138.402,A -85,B 0,C 180,E1 -11824.669,E2 -11824.669} C_VEL
LIN {X 0,Y 382.991,Z 138.407,A -85,B 0,C 180,E1 -11827.902,E2 -11827.902} C_VEL
LIN {X 0,Y 382.961,Z 138.41,A -85,B 0,C 180,E1 -11831.351,E2 -11831.351} C_VEL
LIN {X 0,Y 382.989,Z 138.402,A -85,B 0,C 180,E1 -11834.302,E2 -11834.302} C_VEL
LIN {X 0,Y 382.983,Z 138.391,A -85,B 0,C 180,E1 -11837.236,E2 -11837.236} C_VEL
LIN {X 0,Y 382.986,Z 138.405,A -85,B 0,C 180,E1 -11840.419,E2 -11840.419} C_VEL
LIN {X 0,Y 383.014,Z 138.391,A -85,B 0,C 180,E1 -11844.043,E2 -11844.043} C_VEL
LIN {X 0,Y 382.984,Z 138.393,A -85,B 0,C 180,E1 -11847.579,E2 -11847.579} C_VEL
LIN {X 0,Y 382.975,Z 138.393,A -85,B 0,C 180,E1 -11850.299,E2 -11850.299} C_VEL
LIN {X 0,Y 383.004,Z 138.397,A -85,B 0,C 180,E1 -11854.045,E2 -11854.045} C_VEL
LIN {X 0,Y 382.99,Z 138.397,A -85,B 0,C 180,E1 -11857.334,E2 -11857.334} C_VEL
LIN {X 0,Y 383.044,Z 138.393,A -85,B 0,C 180,E1 -11860.715,E2 -11860.715} C_VEL
LIN {X 0,Y 383.023,Z 138.401,A -85,B 0,C 180,E1 -11864.024,E2 -11864.024} C_VEL
LIN {X 0,Y 383.139,Z 138.379,A -85,B 0,C 180,E1 -11867.284,E2 -11867.284} C_VEL
LIN {X 0,Y 383.145,Z 138.374,A -85,B 0,C 180,E1 -11870.498,E2 -11870.498} C_VEL
LIN {X 0,Y 383.236,Z 138.374,A -85,B 0,C 180,E1 -11873.683,E2 -11873.683} C_VEL
LIN {X 0,Y 383.376,Z 138.356,A -85,B 0,C 180,E1 -11877.899,E2 -11877.899} C_VEL
LIN {X 0,Y 383.265,Z 138.363,A -85,B 0,C 180,E1 -11881.051,E2 -11881.051} C_VEL
LIN {X 0,Y 383.238,Z 138.373,A -85,B 0,C 180,E1 -11883.154,E2 -11883.154} C_VEL
LIN {X 0,Y 383.245,Z 138.369,A -85,B 0,C 180,E1 -11886.317,E2 -11886.317} C_VEL
LIN {X 0,Y 383.146,Z 138.379,A -85,B 0,C 180,E1 -11889.502,E2 -11889.502} C_VEL
LIN {X 0,Y 383.139,Z 138.384,A -85,B 0,C 180,E1 -11892.716,E2 -11892.716} C_VEL
LIN {X 0,Y 383.082,Z 138.392,A -85,B 0,C 180,E1 -11895.973,E2 -11895.973} C_VEL
LIN {X 0,Y 383.061,Z 138.395,A -85,B 0,C 180,E1 -11899.284,E2 -11899.284} C_VEL
LIN {X 0,Y 382.999,Z 138.397,A -85,B 0,C 180,E1 -11902.665,E2 -11902.665} C_VEL
LIN {X 0,Y 383.039,Z 138.393,A -85,B 0,C 180,E1 -11906.126,E2 -11906.126} C_VEL
LIN {X 0,Y 382.986,Z 138.402,A -85,B 0,C 180,E1 -11909.7,E2 -11909.7} C_VEL
LIN {X 0,Y 383.004,Z 138.394,A -85,B 0,C 180,E1 -11913.4,E2 -11913.4} C_VEL
LIN {X 0,Y 383.033,Z 138.398,A -85,B 0,C 180,E1 -11916.164,E2 -11916.164} C_VEL
LIN {X 0,Y 383.009,Z 138.397,A -85,B 0,C 180,E1 -11919.958,E2 -11919.958} C_VEL
LIN {X 0,Y 383.006,Z 138.4,A -85,B 0,C 180,E1 -11922.778,E2 -11922.778} C_VEL
LIN {X 0,Y 382.998,Z 138.402,A -85,B 0,C 180,E1 -11925.789,E2 -11925.789} C_VEL
LIN {X 0,Y 382.989,Z 138.397,A -85,B 0,C 180,E1 -11928.796,E2 -11928.796} C_VEL
LIN {X 0,Y 383.001,Z 138.399,A -85,B 0,C 180,E1 -11932.096,E2 -11932.096} C_VEL
LIN {X 0,Y 383.068,Z 138.523,A -85,B 0,C 180,E1 -11934.615,E2 -11934.615} C_VEL
LIN {X 0,Y 386.92,Z 153.096,A -85,B 0,C 180,E1 -11937.907,E2 -11937.907} C_VEL
LIN {X 0,Y 389.636,Z 164.569,A -85,B 0,C 180,E1 -11940.357,E2 -11940.357} C_VEL
LIN {X 0,Y 392.582,Z 171.819,A -85,B 0,C 180,E1 -11940.756,E2 -11940.756} C_VEL
LIN {X 0,Y 398.3,Z 200.858,A -85,B 0,C 180,E1 -11941.794,E2 -11941.794} C_VEL
LIN {X 0,Y 398.832,Z 204.509,A -85,B 0,C 180,E1 -11941.908,E2 -11941.908} C_VEL
LIN {X 0,Y 396.278,Z 322.884,A -85,B 0,C 180,E1 -11944.069,E2 -11944.069} C_VEL
LIN {X 0,Y 395.649,Z 338.636,A -85,B 0,C 180,E1 -11944.449,E2 -11944.449} C_VEL
LIN {X 0,Y 394.552,Z 354.455,A -85,B 0,C 180,E1 -11945.043,E2 -11945.043} C_VEL
LIN {X 0,Y 393.404,Z 368.715,A -85,B 0,C 180,E1 -11945.793,E2 -11945.793} C_VEL
LIN {X 0,Y 391.932,Z 383.077,A -85,B 0,C 180,E1 -11946.765,E2 -11946.765} C_VEL
LIN {X 0,Y 390.329,Z 396.684,A -85,B 0,C 180,E1 -11947.922,E2 -11947.922} C_VEL
LIN {X 0,Y 388.731,Z 409.122,A -85,B 0,C 180,E1 -11949.218,E2 -11949.218} C_VEL
LIN {X 0,Y 387.292,Z 420.64,A -85,B 0,C 180,E1 -11950.668,E2 -11950.668} C_VEL
LIN {X 0,Y 385.904,Z 431.122,A -85,B 0,C 180,E1 -11952.239,E2 -11952.239} C_VEL
LIN {X 0,Y 384.658,Z 440.067,A -85,B 0,C 180,E1 -11953.821,E2 -11953.821} C_VEL
LIN {X 0,Y 383.579,Z 448.88,A -85,B 0,C 180,E1 -11955.679,E2 -11955.679} C_VEL
LIN {X 0,Y 382.899,Z 455.263,A -85,B 0,C 180,E1 -11957.276,E2 -11957.276} C_VEL
LIN {X 0,Y 382.185,Z 462.271,A -85,B 0,C 180,E1 -11959.403,E2 -11959.403} C_VEL
LIN {X 0,Y 381.828,Z 467.786,A -85,B 0,C 180,E1 -11961.532,E2 -11961.532} C_VEL
LIN {X 0,Y 381.653,Z 472.419,A -85,B 0,C 180,E1 -11963.927,E2 -11963.927} C_VEL
LIN {X 0,Y 381.574,Z 474.882,A -85,B 0,C 180,E1 -11965.775,E2 -11965.775} C_VEL
LIN {X 0,Y 381.551,Z 476.626,A -85,B 0,C 180,E1 -11967.889,E2 -11967.889} C_VEL
LIN {X 0,Y 381.636,Z 477.226,A -85,B 0,C 180,E1 -11970,E2 -11970} C_VEL
LIN {X 0,Y 381.551,Z 476.62,A -85,B 0,C 180,E1 -11972.111,E2 -11972.111} C_VEL
LIN {X 0,Y 381.576,Z 474.868,A -85,B 0,C 180,E1 -11974.225,E2 -11974.225} C_VEL
LIN {X 0,Y 381.664,Z 471.941,A -85,B 0,C 180,E1 -11976.343,E2 -11976.343} C_VEL
LIN {X 0,Y 381.828,Z 467.769,A -85,B 0,C 180,E1 -11978.468,E2 -11978.468} C_VEL
LIN {X 0,Y 382.183,Z 462.244,A -85,B 0,C 180,E1 -11980.596,E2 -11980.596} C_VEL
LIN {X 0,Y 382.897,Z 455.221,A -85,B 0,C 180,E1 -11982.724,E2 -11982.724} C_VEL
LIN {X 0,Y 383.703,Z 447.708,A -85,B 0,C 180,E1 -11984.587,E2 -11984.587} C_VEL
LIN {X 0,Y 384.827,Z 438.655,A -85,B 0,C 180,E1 -11986.444,E2 -11986.444} C_VEL
LIN {X 0,Y 386.34,Z 427.784,A -85,B 0,C 180,E1 -11988.288,E2 -11988.288} C_VEL
LIN {X 0,Y 387.856,Z 415.668,A -85,B 0,C 180,E1 -11989.986,E2 -11989.986} C_VEL
LIN {X 0,Y 389.519,Z 403.103,A -85,B 0,C 180,E1 -11991.43,E2 -11991.43} C_VEL
LIN {X 0,Y 391.011,Z 390.849,A -85,B 0,C 180,E1 -11992.594,E2 -11992.594} C_VEL
LIN {X 0,Y 392.502,Z 377.616,A -85,B 0,C 180,E1 -11993.618,E2 -11993.618} C_VEL
LIN {X 0,Y 393.927,Z 362.581,A -85,B 0,C 180,E1 -11994.542,E2 -11994.542} C_VEL
LIN {X 0,Y 395.071,Z 347.474,A -85,B 0,C 180,E1 -11995.235,E2 -11995.235} C_VEL
LIN {X 0,Y 395.913,Z 332.563,A -85,B 0,C 180,E1 -11995.709,E2 -11995.709} C_VEL
LIN {X 0,Y 396.741,Z 298.994,A -85,B 0,C 180,E1 -11996.357,E2 -11996.357} C_VEL
LIN {X 0,Y 398.768,Z 203.675,A -85,B 0,C 180,E1 -11998.101,E2 -11998.101} C_VEL
LIN {X 0,Y 394.111,Z 179.375,A -85,B 0,C 180,E1 -11998.953,E2 -11998.953} C_VEL
LIN {X 0,Y 392.041,Z 170.342,A -85,B 0,C 180,E1 -11999.304,E2 -11999.304} C_VEL
LIN {X 0,Y 389.615,Z 164.514,A -85,B 0,C 180,E1 -11999.64,E2 -11999.64} C_VEL
LIN {X 0,Y 386.48,Z 151.435,A -85,B 0,C 180,E1 -12002.442,E2 -12002.442} C_VEL
LIN {X 0,Y 383.028,Z 138.397,A -85,B 0,C 180,E1 -12005.429,E2 -12005.429} C_VEL
LIN {X 0,Y 383.006,Z 138.401,A -85,B 0,C 180,E1 -12008.601,E2 -12008.601} C_VEL
LIN {X 0,Y 382.985,Z 138.403,A -85,B 0,C 180,E1 -12011.347,E2 -12011.347} C_VEL
LIN {X 0,Y 382.996,Z 138.399,A -85,B 0,C 180,E1 -12014.304,E2 -12014.304} C_VEL
LIN {X 0,Y 383.011,Z 138.398,A -85,B 0,C 180,E1 -12017.24,E2 -12017.24} C_VEL
LIN {X 0,Y 383.014,Z 138.397,A -85,B 0,C 180,E1 -12020.414,E2 -12020.414} C_VEL
LIN {X 0,Y 383.025,Z 138.392,A -85,B 0,C 180,E1 -12024.045,E2 -12024.045} C_VEL
LIN {X 0,Y 382.988,Z 138.401,A -85,B 0,C 180,E1 -12027.578,E2 -12027.578} C_VEL
LIN {X 0,Y 382.993,Z 138.396,A -85,B 0,C 180,E1 -12030.3,E2 -12030.3} C_VEL
LIN {X 0,Y 383.057,Z 138.393,A -85,B 0,C 180,E1 -12032.698,E2 -12032.698} C_VEL
LIN {X 0,Y 383.05,Z 138.398,A -85,B 0,C 180,E1 -12035.04,E2 -12035.04} C_VEL
LIN {X 0,Y 382.994,Z 138.402,A -85,B 0,C 180,E1 -12038.469,E2 -12038.469} C_VEL
LIN {X 0,Y 383.063,Z 138.392,A -85,B 0,C 180,E1 -12041.827,E2 -12041.827} C_VEL
LIN {X 0,Y 383.112,Z 138.389,A -85,B 0,C 180,E1 -12045.118,E2 -12045.118} C_VEL
LIN {X 0,Y 383.099,Z 138.384,A -85,B 0,C 180,E1 -12048.358,E2 -12048.358} C_VEL
LIN {X 0,Y 383.217,Z 138.367,A -85,B 0,C 180,E1 -12052.028,E2 -12052.028} C_VEL
LIN {X 0,Y 383.184,Z 138.376,A -85,B 0,C 180,E1 -12054.738,E2 -12054.738} C_VEL
LIN {X 0,Y 383.385,Z 138.353,A -85,B 0,C 180,E1 -12057.899,E2 -12057.899} C_VEL
LIN {X 0,Y 383.302,Z 138.361,A -85,B 0,C 180,E1 -12061.051,E2 -12061.051} C_VEL
LIN {X 0,Y 383.202,Z 138.374,A -85,B 0,C 180,E1 -12063.154,E2 -12063.154} C_VEL
LIN {X 0,Y 383.233,Z 138.374,A -85,B 0,C 180,E1 -12066.43,E2 -12066.43} C_VEL
LIN {X 0,Y 383.144,Z 138.376,A -85,B 0,C 180,E1 -12069.502,E2 -12069.502} C_VEL
LIN {X 0,Y 383.128,Z 138.379,A -85,B 0,C 180,E1 -12073.536,E2 -12073.536} C_VEL
LIN {X 0,Y 383.06,Z 138.388,A -85,B 0,C 180,E1 -12077.437,E2 -12077.437} C_VEL
LIN {X 0,Y 383.031,Z 138.392,A -85,B 0,C 180,E1 -12080.647,E2 -12080.647} C_VEL
LIN {X 0,Y 383.011,Z 138.399,A -85,B 0,C 180,E1 -12083.809,E2 -12083.809} C_VEL
LIN {X 0,Y 382.972,Z 138.386,A -85,B 0,C 180,E1 -12087.309,E2 -12087.309} C_VEL
LIN {X 0,Y 382.983,Z 138.402,A -85,B 0,C 180,E1 -12090.919,E2 -12090.919} C_VEL
LIN {X 0,Y 383.018,Z 138.393,A -85,B 0,C 180,E1 -12094.668,E2 -12094.668} C_VEL
LIN {X 0,Y 382.994,Z 138.4,A -85,B 0,C 180,E1 -12097.902,E2 -12097.902} C_VEL
LIN {X 0,Y 382.961,Z 138.405,A -85,B 0,C 180,E1 -12101.351,E2 -12101.351} C_VEL
LIN {X 0,Y 382.99,Z 138.399,A -85,B 0,C 180,E1 -12104.302,E2 -12104.302} C_VEL
LIN {X 0,Y 382.997,Z 138.403,A -85,B 0,C 180,E1 -12107.238,E2 -12107.238} C_VEL
LIN {X 0,Y 382.985,Z 138.403,A -85,B 0,C 180,E1 -12110.419,E2 -12110.419} C_VEL
LIN {X 0,Y 383.013,Z 138.396,A -85,B 0,C 180,E1 -12114.043,E2 -12114.043} C_VEL
LIN {X 0,Y 382.982,Z 138.402,A -85,B 0,C 180,E1 -12117.58,E2 -12117.58} C_VEL
LIN {X 0,Y 383.01,Z 138.521,A -85,B 0,C 180,E1 -12118.121,E2 -12118.121} C_VEL
LIN {X 0,Y 385.112,Z 146.542,A -85,B 0,C 180,E1 -12120.058,E2 -12120.058} C_VEL
LIN {X 0,Y 395.32,Z 168.561,A -85,B 0,C 180,E1 -12121.362,E2 -12121.362} C_VEL
LIN {X 0,Y 399.223,Z 178.197,A -85,B 0,C 180,E1 -12121.864,E2 -12121.864} C_VEL
LIN {X 0,Y 397.425,Z 264.289,A -85,B 0,C 180,E1 -12123.444,E2 -12123.444} C_VEL
LIN {X 0,Y 396.303,Z 311.078,A -85,B 0,C 180,E1 -12124.318,E2 -12124.318} C_VEL
LIN {X 0,Y 395.649,Z 325.986,A -85,B 0,C 180,E1 -12124.786,E2 -12124.786} C_VEL
LIN {X 0,Y 394.706,Z 340.989,A -85,B 0,C 180,E1 -12125.466,E2 -12125.466} C_VEL
LIN {X 0,Y 393.515,Z 354.999,A -85,B 0,C 180,E1 -12126.307,E2 -12126.307} C_VEL
LIN {X 0,Y 392.08,Z 368.579,A -85,B 0,C 180,E1 -12127.332,E2 -12127.332} C_VEL
LIN {X 0,Y 390.431,Z 382.353,A -85,B 0,C 180,E1 -12128.622,E2 -12128.622} C_VEL
LIN {X 0,Y 388.875,Z 394.462,A -85,B 0,C 180,E1 -12130.014,E2 -12130.014} C_VEL
LIN {X 0,Y 387.47,Z 405.169,A -85,B 0,C 180,E1 -12131.493,E2 -12131.493} C_VEL
LIN {X 0,Y 386.185,Z 414.809,A -85,B 0,C 180,E1 -12133.072,E2 -12133.072} C_VEL
LIN {X 0,Y 384.843,Z 424.258,A -85,B 0,C 180,E1 -12134.916,E2 -12134.916} C_VEL
LIN {X 0,Y 383.916,Z 432.117,A -85,B 0,C 180,E1 -12136.772,E2 -12136.772} C_VEL
LIN {X 0,Y 382.938,Z 439.457,A -85,B 0,C 180,E1 -12138.889,E2 -12138.889} C_VEL
LIN {X 0,Y 382.365,Z 445.275,A -85,B 0,C 180,E1 -12141.012,E2 -12141.012} C_VEL
LIN {X 0,Y 382.058,Z 448.719,A -85,B 0,C 180,E1 -12142.602,E2 -12142.602} C_VEL
LIN {X 0,Y 381.816,Z 452.209,A -85,B 0,C 180,E1 -12144.719,E2 -12144.719} C_VEL
LIN {X 0,Y 381.619,Z 454.682,A -85,B 0,C 180,E1 -12147.071,E2 -12147.071} C_VEL
LIN {X 0,Y 381.64,Z 455.696,A -85,B 0,C 180,E1 -12148.945,E2 -12148.945} C_VEL
LIN {X 0,Y 381.641,Z 455.711,A -85,B 0,C 180,E1 -12151.055,E2 -12151.055} C_VEL
LIN {X 0,Y 381.624,Z 455.473,A -85,B 0,C 180,E1 -12151.656,E2 -12151.656} C_VEL
LIN {X 0,Y 380.969,Z 455.091,A -85,B 0,C 180,E1 -12152.535,E2 -12152.535} C_VEL
LIN {X 0,Y 378.148,Z 454.031,A -85,B 0,C 180,E1 -12153.96,E2 -12153.96} C_VEL
LIN {X 0,Y 375.807,Z 452.864,A -85,B 0,C 180,E1 -12155.105,E2 -12155.105} C_VEL
LIN {X 0,Y 374.833,Z 451.519,A -85,B 0,C 180,E1 -12156.132,E2 -12156.132} C_VEL
LIN {X 0,Y 374.835,Z 451.242,A -85,B 0,C 180,E1 -12156.28,E2 -12156.28} C_VEL
LIN {X 0,Y 375.177,Z 446.929,A -85,B 0,C 180,E1 -12158.619,E2 -12158.619} C_VEL
LIN {X 0,Y 375.752,Z 441.551,A -85,B 0,C 180,E1 -12160.78,E2 -12160.78} C_VEL
LIN {X 0,Y 376.687,Z 434.692,A -85,B 0,C 180,E1 -12162.938,E2 -12162.938} C_VEL
LIN {X 0,Y 377.585,Z 427.206,A -85,B 0,C 180,E1 -12164.857,E2 -12164.857} C_VEL
LIN {X 0,Y 378.842,Z 418.431,A -85,B 0,C 180,E1 -12166.711,E2 -12166.711} C_VEL
LIN {X 0,Y 380.151,Z 409.365,A -85,B 0,C 180,E1 -12168.318,E2 -12168.318} C_VEL
LIN {X 0,Y 381.827,Z 398.068,A -85,B 0,C 180,E1 -12169.995,E2 -12169.995} C_VEL
LIN {X 0,Y 383.41,Z 385.815,A -85,B 0,C 180,E1 -12171.507,E2 -12171.507} C_VEL
LIN {X 0,Y 385.076,Z 372.8,A -85,B 0,C 180,E1 -12172.82,E2 -12172.82} C_VEL
LIN {X 0,Y 386.559,Z 360.129,A -85,B 0,C 180,E1 -12173.862,E2 -12173.862} C_VEL
LIN {X 0,Y 387.804,Z 347.126,A -85,B 0,C 180,E1 -12174.731,E2 -12174.731} C_VEL
LIN {X 0,Y 388.847,Z 332.723,A -85,B 0,C 180,E1 -12175.485,E2 -12175.485} C_VEL
LIN {X 0,Y 389.719,Z 318.01,A -85,B 0,C 180,E1 -12176.04,E2 -12176.04} C_VEL
LIN {X 0,Y 390.247,Z 303.587,A -85,B 0,C 180,E1 -12176.398,E2 -12176.398} C_VEL
LIN {X 0,Y 393.018,Z 181.167,A -85,B 0,C 180,E1 -12178.669,E2 -12178.669} C_VEL
LIN {X 0,Y 392.581,Z 178.869,A -85,B 0,C 180,E1 -12178.751,E2 -12178.751} C_VEL
LIN {X 0,Y 383.423,Z 158.098,A -85,B 0,C 180,E1 -12179.95,E2 -12179.95} C_VEL
LIN {X 0,Y 377.819,Z 146.465,A -85,B 0,C 180,E1 -12180.713,E2 -12180.713} C_VEL
LIN {X 0,Y 375.945,Z 139.284,A -85,B 0,C 180,E1 -12182.57,E2 -12182.57} C_VEL
LIN {X 0,Y 375.948,Z 139.286,A -85,B 0,C 180,E1 -12185.417,E2 -12185.417} C_VEL
LIN {X 0,Y 375.933,Z 139.286,A -85,B 0,C 180,E1 -12188.262,E2 -12188.262} C_VEL
LIN {X 0,Y 375.914,Z 139.286,A -85,B 0,C 180,E1 -12191.597,E2 -12191.597} C_VEL
LIN {X 0,Y 375.921,Z 139.283,A -85,B 0,C 180,E1 -12194.73,E2 -12194.73} C_VEL
LIN {X 0,Y 375.908,Z 139.271,A -85,B 0,C 180,E1 -12197.696,E2 -12197.696} C_VEL
LIN {X 0,Y 375.935,Z 139.283,A -85,B 0,C 180,E1 -12200.534,E2 -12200.534} C_VEL
LIN {X 0,Y 375.958,Z 139.267,A -85,B 0,C 180,E1 -12203.497,E2 -12203.497} C_VEL
LIN {X 0,Y 375.959,Z 139.278,A -85,B 0,C 180,E1 -12205.888,E2 -12205.888} C_VEL
LIN {X 0,Y 375.961,Z 139.263,A -85,B 0,C 180,E1 -12209.687,E2 -12209.687} C_VEL
LIN {X 0,Y 375.919,Z 139.285,A -85,B 0,C 180,E1 -12212.135,E2 -12212.135} C_VEL
LIN {X 0,Y 375.937,Z 139.279,A -85,B 0,C 180,E1 -12214.534,E2 -12214.534} C_VEL
LIN {X 0,Y 375.976,Z 139.272,A -85,B 0,C 180,E1 -12216.887,E2 -12216.887} C_VEL
LIN {X 0,Y 375.989,Z 139.275,A -85,B 0,C 180,E1 -12220.339,E2 -12220.339} C_VEL
LIN {X 0,Y 375.978,Z 139.276,A -85,B 0,C 180,E1 -12223.716,E2 -12223.716} C_VEL
LIN {X 0,Y 376.106,Z 139.255,A -85,B 0,C 180,E1 -12227.042,E2 -12227.042} C_VEL
LIN {X 0,Y 376.115,Z 139.251,A -85,B 0,C 180,E1 -12230.318,E2 -12230.318} C_VEL
LIN {X 0,Y 376.196,Z 139.251,A -85,B 0,C 180,E1 -12233.564,E2 -12233.564} C_VEL
LIN {X 0,Y 376.34,Z 139.233,A -85,B 0,C 180,E1 -12237.859,E2 -12237.859} C_VEL
LIN {X 0,Y 376.236,Z 139.238,A -85,B 0,C 180,E1 -12241.07,E2 -12241.07} C_VEL
LIN {X 0,Y 376.351,Z 139.23,A -85,B 0,C 180,E1 -12242.14,E2 -12242.14} C_VEL
LIN {X 0,Y 376.203,Z 139.246,A -85,B 0,C 180,E1 -12246.436,E2 -12246.436} C_VEL
LIN {X 0,Y 376.116,Z 139.255,A -85,B 0,C 180,E1 -12249.681,E2 -12249.681} C_VEL
LIN {X 0,Y 376.092,Z 139.256,A -85,B 0,C 180,E1 -12253.657,E2 -12253.657} C_VEL
LIN {X 0,Y 376.035,Z 139.265,A -85,B 0,C 180,E1 -12257.4,E2 -12257.4} C_VEL
LIN {X 0,Y 375.98,Z 139.281,A -85,B 0,C 180,E1 -12260.832,E2 -12260.832} C_VEL
LIN {X 0,Y 375.985,Z 139.276,A -85,B 0,C 180,E1 -12264.282,E2 -12264.282} C_VEL
LIN {X 0,Y 375.966,Z 139.273,A -85,B 0,C 180,E1 -12266.656,E2 -12266.656} C_VEL
LIN {X 0,Y 375.964,Z 139.279,A -85,B 0,C 180,E1 -12270.313,E2 -12270.313} C_VEL
LIN {X 0,Y 375.961,Z 139.271,A -85,B 0,C 180,E1 -12274.111,E2 -12274.111} C_VEL
LIN {X 0,Y 375.954,Z 139.275,A -85,B 0,C 180,E1 -12276.741,E2 -12276.741} C_VEL
LIN {X 0,Y 375.989,Z 139.271,A -85,B 0,C 180,E1 -12279.97,E2 -12279.97} C_VEL
LIN {X 0,Y 375.931,Z 139.283,A -85,B 0,C 180,E1 -12283.766,E2 -12283.766} C_VEL
LIN {X 0,Y 375.935,Z 139.279,A -85,B 0,C 180,E1 -12286.81,E2 -12286.81} C_VEL
LIN {X 0,Y 375.964,Z 139.268,A -85,B 0,C 180,E1 -12290.537,E2 -12290.537} C_VEL
LIN {X 0,Y 375.987,Z 139.284,A -85,B 0,C 180,E1 -12294.052,E2 -12294.052} C_VEL
LIN {X 0,Y 379.385,Z 152.077,A -85,B 0,C 180,E1 -12297.031,E2 -12297.031} C_VEL
LIN {X 0,Y 382.398,Z 164.385,A -85,B 0,C 180,E1 -12299.746,E2 -12299.746} C_VEL
LIN {X 0,Y 386.748,Z 174.92,A -85,B 0,C 180,E1 -12300.339,E2 -12300.339} C_VEL
LIN {X 0,Y 392.193,Z 202.876,A -85,B 0,C 180,E1 -12301.36,E2 -12301.36} C_VEL
LIN {X 0,Y 392.531,Z 207.038,A -85,B 0,C 180,E1 -12301.471,E2 -12301.471} C_VEL
LIN {X 0,Y 389.72,Z 328.833,A -85,B 0,C 180,E1 -12303.744,E2 -12303.744} C_VEL
LIN {X 0,Y 389.001,Z 343.085,A -85,B 0,C 180,E1 -12304.16,E2 -12304.16} C_VEL
LIN {X 0,Y 387.793,Z 358.179,A -85,B 0,C 180,E1 -12304.793,E2 -12304.793} C_VEL
LIN {X 0,Y 386.549,Z 372.357,A -85,B 0,C 180,E1 -12305.608,E2 -12305.608} C_VEL
LIN {X 0,Y 385.012,Z 386.087,A -85,B 0,C 180,E1 -12306.608,E2 -12306.608} C_VEL
LIN {X 0,Y 383.4,Z 399.114,A -85,B 0,C 180,E1 -12307.786,E2 -12307.786} C_VEL
LIN {X 0,Y 381.721,Z 411.145,A -85,B 0,C 180,E1 -12309.101,E2 -12309.101} C_VEL
LIN {X 0,Y 380.269,Z 422.296,A -85,B 0,C 180,E1 -12310.569,E2 -12310.569} C_VEL
LIN {X 0,Y 378.84,Z 432.559,A -85,B 0,C 180,E1 -12312.176,E2 -12312.176} C_VEL
LIN {X 0,Y 377.421,Z 442.592,A -85,B 0,C 180,E1 -12314.058,E2 -12314.058} C_VEL
LIN {X 0,Y 376.306,Z 450.928,A -85,B 0,C 180,E1 -12315.949,E2 -12315.949} C_VEL
LIN {X 0,Y 375.558,Z 458.769,A -85,B 0,C 180,E1 -12318.121,E2 -12318.121} C_VEL
LIN {X 0,Y 374.926,Z 465.005,A -85,B 0,C 180,E1 -12320.287,E2 -12320.287} C_VEL
LIN {X 0,Y 374.653,Z 469.834,A -85,B 0,C 180,E1 -12322.455,E2 -12322.455} C_VEL
LIN {X 0,Y 374.489,Z 473.371,A -85,B 0,C 180,E1 -12324.616,E2 -12324.616} C_VEL
LIN {X 0,Y 374.435,Z 475.699,A -85,B 0,C 180,E1 -12326.772,E2 -12326.772} C_VEL
LIN {X 0,Y 374.514,Z 476.872,A -85,B 0,C 180,E1 -12328.925,E2 -12328.925} C_VEL
LIN {X 0,Y 374.514,Z 476.87,A -85,B 0,C 180,E1 -12331.075,E2 -12331.075} C_VEL
LIN {X 0,Y 374.436,Z 475.688,A -85,B 0,C 180,E1 -12333.228,E2 -12333.228} C_VEL
LIN {X 0,Y 374.494,Z 473.354,A -85,B 0,C 180,E1 -12335.384,E2 -12335.384} C_VEL
LIN {X 0,Y 374.653,Z 469.816,A -85,B 0,C 180,E1 -12337.545,E2 -12337.545} C_VEL
LIN {X 0,Y 374.926,Z 464.983,A -85,B 0,C 180,E1 -12339.713,E2 -12339.713} C_VEL
LIN {X 0,Y 375.551,Z 458.731,A -85,B 0,C 180,E1 -12341.879,E2 -12341.879} C_VEL
LIN {X 0,Y 376.306,Z 450.879,A -85,B 0,C 180,E1 -12344.051,E2 -12344.051} C_VEL
LIN {X 0,Y 377.419,Z 442.538,A -85,B 0,C 180,E1 -12345.942,E2 -12345.942} C_VEL
LIN {X 0,Y 378.8,Z 432.493,A -85,B 0,C 180,E1 -12347.826,E2 -12347.826} C_VEL
LIN {X 0,Y 380.269,Z 421.682,A -85,B 0,C 180,E1 -12349.513,E2 -12349.513} C_VEL
LIN {X 0,Y 381.888,Z 409.988,A -85,B 0,C 180,E1 -12351.031,E2 -12351.031} C_VEL
LIN {X 0,Y 383.511,Z 397.712,A -85,B 0,C 180,E1 -12352.349,E2 -12352.349} C_VEL
LIN {X 0,Y 385.178,Z 384.356,A -85,B 0,C 180,E1 -12353.524,E2 -12353.524} C_VEL
LIN {X 0,Y 386.702,Z 370.611,A -85,B 0,C 180,E1 -12354.494,E2 -12354.494} C_VEL
LIN {X 0,Y 387.983,Z 356.13,A -85,B 0,C 180,E1 -12355.294,E2 -12355.294} C_VEL
LIN {X 0,Y 389.065,Z 340.936,A -85,B 0,C 180,E1 -12355.907,E2 -12355.907} C_VEL
LIN {X 0,Y 389.823,Z 325.277,A -85,B 0,C 180,E1 -12356.321,E2 -12356.321} C_VEL
LIN {X 0,Y 392.519,Z 205.34,A -85,B 0,C 180,E1 -12358.551,E2 -12358.551} C_VEL
LIN {X 0,Y 388.136,Z 181.758,A -85,B 0,C 180,E1 -12359.388,E2 -12359.388} C_VEL
LIN {X 0,Y 386.166,Z 173.133,A -85,B 0,C 180,E1 -12359.732,E2 -12359.732} C_VEL
LIN {X 0,Y 382.403,Z 164.286,A -85,B 0,C 180,E1 -12360.255,E2 -12360.255} C_VEL
LIN {X 0,Y 378.887,Z 150.017,A -85,B 0,C 180,E1 -12363.415,E2 -12363.415} C_VEL
LIN {X 0,Y 375.987,Z 139.272,A -85,B 0,C 180,E1 -12365.948,E2 -12365.948} C_VEL
LIN {X 0,Y 375.964,Z 139.278,A -85,B 0,C 180,E1 -12369.463,E2 -12369.463} C_VEL
LIN {X 0,Y 375.935,Z 139.28,A -85,B 0,C 180,E1 -12373.19,E2 -12373.19} C_VEL
LIN {X 0,Y 375.934,Z 139.278,A -85,B 0,C 180,E1 -12376.811,E2 -12376.811} C_VEL
LIN {X 0,Y 375.962,Z 139.276,A -85,B 0,C 180,E1 -12380.537,E2 -12380.537} C_VEL
LIN {X 0,Y 375.964,Z 139.275,A -85,B 0,C 180,E1 -12383.496,E2 -12383.496} C_VEL
LIN {X 0,Y 375.961,Z 139.275,A -85,B 0,C 180,E1 -12385.889,E2 -12385.889} C_VEL
LIN {X 0,Y 375.966,Z 139.272,A -85,B 0,C 180,E1 -12389.688,E2 -12389.688} C_VEL
LIN {X 0,Y 375.997,Z 139.271,A -85,B 0,C 180,E1 -12392.142,E2 -12392.142} C_VEL
LIN {X 0,Y 376.005,Z 139.271,A -85,B 0,C 180,E1 -12394.539,E2 -12394.539} C_VEL
LIN {X 0,Y 375.958,Z 139.277,A -85,B 0,C 180,E1 -12398.046,E2 -12398.046} C_VEL
LIN {X 0,Y 376.009,Z 139.272,A -85,B 0,C 180,E1 -12401.473,E2 -12401.473} C_VEL
LIN {X 0,Y 376.06,Z 139.265,A -85,B 0,C 180,E1 -12404.833,E2 -12404.833} C_VEL
LIN {X 0,Y 376.051,Z 139.26,A -85,B 0,C 180,E1 -12408.137,E2 -12408.137} C_VEL
LIN {X 0,Y 376.189,Z 139.242,A -85,B 0,C 180,E1 -12411.954,E2 -12411.954} C_VEL
LIN {X 0,Y 376.155,Z 139.253,A -85,B 0,C 180,E1 -12414.64,E2 -12414.64} C_VEL
LIN {X 0,Y 376.351,Z 139.229,A -85,B 0,C 180,E1 -12417.86,E2 -12417.86} C_VEL
LIN {X 0,Y 376.27,Z 139.237,A -85,B 0,C 180,E1 -12421.07,E2 -12421.07} C_VEL
LIN {X 0,Y 376.341,Z 139.232,A -85,B 0,C 180,E1 -12422.141,E2 -12422.141} C_VEL
LIN {X 0,Y 376.202,Z 139.251,A -85,B 0,C 180,E1 -12426.436,E2 -12426.436} C_VEL
LIN {X 0,Y 376.115,Z 139.253,A -85,B 0,C 180,E1 -12429.682,E2 -12429.682} C_VEL
LIN {X 0,Y 376.092,Z 139.256,A -85,B 0,C 180,E1 -12433.658,E2 -12433.658} C_VEL
LIN {X 0,Y 376.014,Z 139.266,A -85,B 0,C 180,E1 -12437.592,E2 -12437.592} C_VEL
LIN {X 0,Y 375.98,Z 139.27,A -85,B 0,C 180,E1 -12440.832,E2 -12440.832} C_VEL
LIN {X 0,Y 375.97,Z 139.271,A -85,B 0,C 180,E1 -12444.283,E2 -12444.283} C_VEL
LIN {X 0,Y 375.919,Z 139.271,A -85,B 0,C 180,E1 -12447.865,E2 -12447.865} C_VEL
LIN {X 0,Y 375.958,Z 139.277,A -85,B 0,C 180,E1 -12451.562,E2 -12451.562} C_VEL
LIN {X 0,Y 375.957,Z 139.279,A -85,B 0,C 180,E1 -12455.416,E2 -12455.416} C_VEL
LIN {X 0,Y 375.936,Z 139.278,A -85,B 0,C 180,E1 -12458.263,E2 -12458.263} C_VEL
LIN {X 0,Y 375.916,Z 139.28,A -85,B 0,C 180,E1 -12461.597,E2 -12461.597} C_VEL
LIN {X 0,Y 375.921,Z 139.281,A -85,B 0,C 180,E1 -12464.73,E2 -12464.73} C_VEL
LIN {X 0,Y 375.917,Z 139.285,A -85,B 0,C 180,E1 -12467.698,E2 -12467.698} C_VEL
LIN {X 0,Y 375.934,Z 139.28,A -85,B 0,C 180,E1 -12470.534,E2 -12470.534} C_VEL
LIN {X 0,Y 375.957,Z 139.279,A -85,B 0,C 180,E1 -12473.497,E2 -12473.497} C_VEL
LIN {X 0,Y 375.958,Z 139.281,A -85,B 0,C 180,E1 -12475.888,E2 -12475.888} C_VEL
LIN {X 0,Y 375.982,Z 139.408,A -85,B 0,C 180,E1 -12477.609,E2 -12477.609} C_VEL
LIN {X 0,Y 377.855,Z 146.574,A -85,B 0,C 180,E1 -12479.417,E2 -12479.417} C_VEL
LIN {X 0,Y 387.525,Z 167.166,A -85,B 0,C 180,E1 -12480.696,E2 -12480.696} C_VEL
LIN {X 0,Y 392.95,Z 179.761,A -85,B 0,C 180,E1 -12481.401,E2 -12481.401} C_VEL
LIN {X 0,Y 391.109,Z 264.513,A -85,B 0,C 180,E1 -12482.981,E2 -12482.981} C_VEL
LIN {X 0,Y 389.939,Z 311.295,A -85,B 0,C 180,E1 -12483.868,E2 -12483.868} C_VEL
LIN {X 0,Y 389.252,Z 326.224,A -85,B 0,C 180,E1 -12484.343,E2 -12484.343} C_VEL
LIN {X 0,Y 388.374,Z 339.838,A -85,B 0,C 180,E1 -12484.964,E2 -12484.964} C_VEL
LIN {X 0,Y 387.212,Z 353.225,A -85,B 0,C 180,E1 -12485.754,E2 -12485.754} C_VEL
LIN {X 0,Y 385.739,Z 367.205,A -85,B 0,C 180,E1 -12486.796,E2 -12486.796} C_VEL
LIN {X 0,Y 384.176,Z 379.983,A -85,B 0,C 180,E1 -12487.974,E2 -12487.974} C_VEL
LIN {X 0,Y 382.454,Z 392.849,A -85,B 0,C 180,E1 -12489.424,E2 -12489.424} C_VEL
LIN {X 0,Y 380.982,Z 403.6,A -85,B 0,C 180,E1 -12490.887,E2 -12490.887} C_VEL
LIN {X 0,Y 379.562,Z 413.537,A -85,B 0,C 180,E1 -12492.489,E2 -12492.489} C_VEL
LIN {X 0,Y 378.131,Z 423.239,A -85,B 0,C 180,E1 -12494.365,E2 -12494.365} C_VEL
LIN {X 0,Y 377.038,Z 431.32,A -85,B 0,C 180,E1 -12496.252,E2 -12496.252} C_VEL
LIN {X 0,Y 376.149,Z 437.986,A -85,B 0,C 180,E1 -12498.14,E2 -12498.14} C_VEL
LIN {X 0,Y 375.455,Z 444.156,A -85,B 0,C 180,E1 -12500.301,E2 -12500.301} C_VEL
LIN {X 0,Y 374.994,Z 448.92,A -85,B 0,C 180,E1 -12502.462,E2 -12502.462} C_VEL
LIN {X 0,Y 374.744,Z 452.409,A -85,B 0,C 180,E1 -12504.619,E2 -12504.619} C_VEL
LIN {X 0,Y 374.538,Z 454.718,A -85,B 0,C 180,E1 -12506.773,E2 -12506.773} C_VEL
LIN {X 0,Y 374.543,Z 455.894,A -85,B 0,C 180,E1 -12508.925,E2 -12508.925} C_VEL
LIN {X 0,Y 374.543,Z 455.91,A -85,B 0,C 180,E1 -12511.075,E2 -12511.075} C_VEL
LIN {X 0,Y 374.537,Z 454.795,A -85,B 0,C 180,E1 -12513.227,E2 -12513.227} C_VEL
LIN {X 0,Y 374.742,Z 452.547,A -85,B 0,C 180,E1 -12515.381,E2 -12515.381} C_VEL
LIN {X 0,Y 374.835,Z 451.242,A -85,B 0,C 180,E1 -12516.28,E2 -12516.28} C_VEL
LIN {X 0,Y 374.309,Z 449.888,A -85,B 0,C 180,E1 -12517.155,E2 -12517.155} C_VEL
LIN {X 0,Y 371.691,Z 447.33,A -85,B 0,C 180,E1 -12518.571,E2 -12518.571} C_VEL
LIN {X 0,Y 369.507,Z 444.978,A -85,B 0,C 180,E1 -12519.698,E2 -12519.698} C_VEL
LIN {X 0,Y 368.686,Z 442.894,A -85,B 0,C 180,E1 -12520.554,E2 -12520.554} C_VEL
LIN {X 0,Y 368.685,Z 442.139,A -85,B 0,C 180,E1 -12520.84,E2 -12520.84} C_VEL
LIN {X 0,Y 369.481,Z 436.723,A -85,B 0,C 180,E1 -12522.635,E2 -12522.635} C_VEL
LIN {X 0,Y 370.47,Z 428.848,A -85,B 0,C 180,E1 -12524.783,E2 -12524.783} C_VEL
LIN {X 0,Y 371.798,Z 419.974,A -85,B 0,C 180,E1 -12526.754,E2 -12526.754} C_VEL
LIN {X 0,Y 373.373,Z 409.562,A -85,B 0,C 180,E1 -12528.663,E2 -12528.663} C_VEL
LIN {X 0,Y 375.055,Z 398.756,A -85,B 0,C 180,E1 -12530.299,E2 -12530.299} C_VEL
LIN {X 0,Y 376.633,Z 387.179,A -85,B 0,C 180,E1 -12531.769,E2 -12531.769} C_VEL
LIN {X 0,Y 378.376,Z 374.414,A -85,B 0,C 180,E1 -12533.103,E2 -12533.103} C_VEL
LIN {X 0,Y 379.884,Z 362.082,A -85,B 0,C 180,E1 -12534.162,E2 -12534.162} C_VEL
LIN {X 0,Y 381.188,Z 348.849,A -85,B 0,C 180,E1 -12535.091,E2 -12535.091} C_VEL
LIN {X 0,Y 382.401,Z 333.8,A -85,B 0,C 180,E1 -12535.904,E2 -12535.904} C_VEL
LIN {X 0,Y 383.297,Z 319.295,A -85,B 0,C 180,E1 -12536.474,E2 -12536.474} C_VEL
LIN {X 0,Y 383.927,Z 303.76,A -85,B 0,C 180,E1 -12536.867,E2 -12536.867} C_VEL
LIN {X 0,Y 386.824,Z 182.322,A -85,B 0,C 180,E1 -12539.151,E2 -12539.151} C_VEL
LIN {X 0,Y 381.125,Z 168.701,A -85,B 0,C 180,E1 -12539.924,E2 -12539.924} C_VEL
LIN {X 0,Y 372.119,Z 149.841,A -85,B 0,C 180,E1 -12541.148,E2 -12541.148} C_VEL
LIN {X 0,Y 370.66,Z 146.694,A -85,B 0,C 180,E1 -12541.371,E2 -12541.371} C_VEL
LIN {X 0,Y 368.91,Z 140.161,A -85,B 0,C 180,E1 -12543.093,E2 -12543.093} C_VEL
LIN {X 0,Y 368.911,Z 140.155,A -85,B 0,C 180,E1 -12546.198,E2 -12546.198} C_VEL
LIN {X 0,Y 368.872,Z 140.159,A -85,B 0,C 180,E1 -12548.957,E2 -12548.957} C_VEL
LIN {X 0,Y 368.859,Z 140.164,A -85,B 0,C 180,E1 -12552.005,E2 -12552.005} C_VEL
LIN {X 0,Y 368.874,Z 140.164,A -85,B 0,C 180,E1 -12555.175,E2 -12555.175} C_VEL
LIN {X 0,Y 368.861,Z 140.15,A -85,B 0,C 180,E1 -12558.174,E2 -12558.174} C_VEL
LIN {X 0,Y 368.877,Z 140.153,A -85,B 0,C 180,E1 -12561.366,E2 -12561.366} C_VEL
LIN {X 0,Y 368.932,Z 140.155,A -85,B 0,C 180,E1 -12565.146,E2 -12565.146} C_VEL
LIN {X 0,Y 368.897,Z 140.137,A -85,B 0,C 180,E1 -12569.043,E2 -12569.043} C_VEL
LIN {X 0,Y 368.908,Z 140.155,A -85,B 0,C 180,E1 -12571.558,E2 -12571.558} C_VEL
LIN {X 0,Y 368.888,Z 140.158,A -85,B 0,C 180,E1 -12575.22,E2 -12575.22} C_VEL
LIN {X 0,Y 368.901,Z 140.152,A -85,B 0,C 180,E1 -12577.603,E2 -12577.603} C_VEL
LIN {X 0,Y 368.923,Z 140.15,A -85,B 0,C 180,E1 -12581.104,E2 -12581.104} C_VEL
LIN {X 0,Y 368.958,Z 140.149,A -85,B 0,C 180,E1 -12584.533,E2 -12584.533} C_VEL
LIN {X 0,Y 369.061,Z 140.133,A -85,B 0,C 180,E1 -12586.79,E2 -12586.79} C_VEL
LIN {X 0,Y 369.065,Z 140.13,A -85,B 0,C 180,E1 -12590.132,E2 -12590.132} C_VEL
LIN {X 0,Y 369.158,Z 140.127,A -85,B 0,C 180,E1 -12593.441,E2 -12593.441} C_VEL
LIN {X 0,Y 369.304,Z 140.11,A -85,B 0,C 180,E1 -12597.819,E2 -12597.819} C_VEL
LIN {X 0,Y 369.207,Z 140.114,A -85,B 0,C 180,E1 -12601.091,E2 -12601.091} C_VEL
LIN {X 0,Y 369.316,Z 140.106,A -85,B 0,C 180,E1 -12602.181,E2 -12602.181} C_VEL
LIN {X 0,Y 369.164,Z 140.124,A -85,B 0,C 180,E1 -12606.559,E2 -12606.559} C_VEL
LIN {X 0,Y 369.066,Z 140.134,A -85,B 0,C 180,E1 -12609.868,E2 -12609.868} C_VEL
LIN {X 0,Y 369.04,Z 140.134,A -85,B 0,C 180,E1 -12613.772,E2 -12613.772} C_VEL
LIN {X 0,Y 368.993,Z 140.14,A -85,B 0,C 180,E1 -12617.743,E2 -12617.743} C_VEL
LIN {X 0,Y 368.912,Z 140.156,A -85,B 0,C 180,E1 -12621.221,E2 -12621.221} C_VEL
LIN {X 0,Y 368.943,Z 140.157,A -85,B 0,C 180,E1 -12624.776,E2 -12624.776} C_VEL
LIN {X 0,Y 368.932,Z 140.156,A -85,B 0,C 180,E1 -12628.44,E2 -12628.44} C_VEL
LIN {X 0,Y 368.903,Z 140.158,A -85,B 0,C 180,E1 -12632.237,E2 -12632.237} C_VEL
LIN {X 0,Y 368.93,Z 140.156,A -85,B 0,C 180,E1 -12635.001,E2 -12635.001} C_VEL
LIN {X 0,Y 368.908,Z 140.158,A -85,B 0,C 180,E1 -12638.64,E2 -12638.64} C_VEL
LIN {X 0,Y 368.882,Z 140.16,A -85,B 0,C 180,E1 -12642.009,E2 -12642.009} C_VEL
LIN {X 0,Y 368.881,Z 140.159,A -85,B 0,C 180,E1 -12645.176,E2 -12645.176} C_VEL
LIN {X 0,Y 368.884,Z 140.16,A -85,B 0,C 180,E1 -12648.177,E2 -12648.177} C_VEL
LIN {X 0,Y 368.91,Z 140.155,A -85,B 0,C 180,E1 -12651.359,E2 -12651.359} C_VEL
LIN {X 0,Y 368.954,Z 140.284,A -85,B 0,C 180,E1 -12653.519,E2 -12653.519} C_VEL
LIN {X 0,Y 372.009,Z 151.543,A -85,B 0,C 180,E1 -12656.227,E2 -12656.227} C_VEL
LIN {X 0,Y 375.19,Z 164.327,A -85,B 0,C 180,E1 -12659.105,E2 -12659.105} C_VEL
LIN {X 0,Y 380.835,Z 177.386,A -85,B 0,C 180,E1 -12659.887,E2 -12659.887} C_VEL
LIN {X 0,Y 386.279,Z 205.917,A -85,B 0,C 180,E1 -12660.946,E2 -12660.946} C_VEL
LIN {X 0,Y 384.077,Z 301.043,A -85,B 0,C 180,E1 -12662.74,E2 -12662.74} C_VEL
LIN {X 0,Y 383.265,Z 331.432,A -85,B 0,C 180,E1 -12663.34,E2 -12663.34} C_VEL
LIN {X 0,Y 382.277,Z 347.333,A -85,B 0,C 180,E1 -12663.858,E2 -12663.858} C_VEL
LIN {X 0,Y 381.072,Z 361.551,A -85,B 0,C 180,E1 -12664.52,E2 -12664.52} C_VEL
LIN {X 0,Y 379.626,Z 376.433,A -85,B 0,C 180,E1 -12665.451,E2 -12665.451} C_VEL
LIN {X 0,Y 377.86,Z 390.574,A -85,B 0,C 180,E1 -12666.574,E2 -12666.574} C_VEL
LIN {X 0,Y 376.043,Z 404.016,A -85,B 0,C 180,E1 -12667.906,E2 -12667.906} C_VEL
LIN {X 0,Y 374.277,Z 416.263,A -85,B 0,C 180,E1 -12669.386,E2 -12669.386} C_VEL
LIN {X 0,Y 372.791,Z 427.576,A -85,B 0,C 180,E1 -12671.043,E2 -12671.043} C_VEL
LIN {X 0,Y 371.067,Z 438.306,A -85,B 0,C 180,E1 -12672.928,E2 -12672.928} C_VEL
LIN {X 0,Y 369.828,Z 447.354,A -85,B 0,C 180,E1 -12674.853,E2 -12674.853} C_VEL
LIN {X 0,Y 368.919,Z 454.864,A -85,B 0,C 180,E1 -12676.785,E2 -12676.785} C_VEL
LIN {X 0,Y 368.139,Z 461.873,A -85,B 0,C 180,E1 -12678.994,E2 -12678.994} C_VEL
LIN {X 0,Y 367.7,Z 467.388,A -85,B 0,C 180,E1 -12681.204,E2 -12681.204} C_VEL
LIN {X 0,Y 367.481,Z 471.559,A -85,B 0,C 180,E1 -12683.411,E2 -12683.411} C_VEL
LIN {X 0,Y 367.387,Z 474.485,A -85,B 0,C 180,E1 -12685.611,E2 -12685.611} C_VEL
LIN {X 0,Y 367.35,Z 476.229,A -85,B 0,C 180,E1 -12687.807,E2 -12687.807} C_VEL
LIN {X 0,Y 367.454,Z 476.829,A -85,B 0,C 180,E1 -12690,E2 -12690} C_VEL
LIN {X 0,Y 367.35,Z 476.222,A -85,B 0,C 180,E1 -12692.193,E2 -12692.193} C_VEL
LIN {X 0,Y 367.389,Z 474.469,A -85,B 0,C 180,E1 -12694.388,E2 -12694.388} C_VEL
LIN {X 0,Y 367.482,Z 471.54,A -85,B 0,C 180,E1 -12696.589,E2 -12696.589} C_VEL
LIN {X 0,Y 367.7,Z 467.367,A -85,B 0,C 180,E1 -12698.795,E2 -12698.795} C_VEL
LIN {X 0,Y 368.136,Z 461.841,A -85,B 0,C 180,E1 -12701.006,E2 -12701.006} C_VEL
LIN {X 0,Y 368.906,Z 454.816,A -85,B 0,C 180,E1 -12703.215,E2 -12703.215} C_VEL
LIN {X 0,Y 369.828,Z 447.302,A -85,B 0,C 180,E1 -12705.147,E2 -12705.147} C_VEL
LIN {X 0,Y 371.05,Z 438.248,A -85,B 0,C 180,E1 -12707.073,E2 -12707.073} C_VEL
LIN {X 0,Y 372.738,Z 427.589,A -85,B 0,C 180,E1 -12708.944,E2 -12708.944} C_VEL
LIN {X 0,Y 374.28,Z 416.18,A -85,B 0,C 180,E1 -12710.614,E2 -12710.614} C_VEL
LIN {X 0,Y 376.036,Z 403.919,A -85,B 0,C 180,E1 -12712.094,E2 -12712.094} C_VEL
LIN {X 0,Y 377.887,Z 390.442,A -85,B 0,C 180,E1 -12713.424,E2 -12713.424} C_VEL
LIN {X 0,Y 379.65,Z 376.142,A -85,B 0,C 180,E1 -12714.557,E2 -12714.557} C_VEL
LIN {X 0,Y 381.116,Z 361.122,A -85,B 0,C 180,E1 -12715.49,E2 -12715.49} C_VEL
LIN {X 0,Y 382.381,Z 345.312,A -85,B 0,C 180,E1 -12716.211,E2 -12716.211} C_VEL
LIN {X 0,Y 383.251,Z 330.989,A -85,B 0,C 180,E1 -12716.661,E2 -12716.661} C_VEL
LIN {X 0,Y 386.089,Z 213.247,A -85,B 0,C 180,E1 -12718.902,E2 -12718.902} C_VEL
LIN {X 0,Y 386.183,Z 205.535,A -85,B 0,C 180,E1 -12719.055,E2 -12719.055} C_VEL
LIN {X 0,Y 381.084,Z 178.75,A -85,B 0,C 180,E1 -12720.046,E2 -12720.046} C_VEL
LIN {X 0,Y 379.974,Z 175.148,A -85,B 0,C 180,E1 -12720.219,E2 -12720.219} C_VEL
LIN {X 0,Y 375.089,Z 163.96,A -85,B 0,C 180,E1 -12720.927,E2 -12720.927} C_VEL
LIN {X 0,Y 372.011,Z 151.441,A -85,B 0,C 180,E1 -12723.773,E2 -12723.773} C_VEL
LIN {X 0,Y 368.931,Z 140.153,A -85,B 0,C 180,E1 -12726.516,E2 -12726.516} C_VEL
LIN {X 0,Y 368.912,Z 140.156,A -85,B 0,C 180,E1 -12730.37,E2 -12730.37} C_VEL
LIN {X 0,Y 368.884,Z 140.163,A -85,B 0,C 180,E1 -12733.616,E2 -12733.616} C_VEL
LIN {X 0,Y 368.886,Z 140.156,A -85,B 0,C 180,E1 -12736.696,E2 -12736.696} C_VEL
LIN {X 0,Y 368.912,Z 140.155,A -85,B 0,C 180,E1 -12739.643,E2 -12739.643} C_VEL
LIN {X 0,Y 368.902,Z 140.157,A -85,B 0,C 180,E1 -12743.145,E2 -12743.145} C_VEL
LIN {X 0,Y 368.897,Z 140.153,A -85,B 0,C 180,E1 -12746.462,E2 -12746.462} C_VEL
LIN {X 0,Y 368.93,Z 140.154,A -85,B 0,C 180,E1 -12749.047,E2 -12749.047} C_VEL
LIN {X 0,Y 368.981,Z 140.147,A -85,B 0,C 180,E1 -12751.564,E2 -12751.564} C_VEL
LIN {X 0,Y 369,Z 140.143,A -85,B 0,C 180,E1 -12754.02,E2 -12754.02} C_VEL
LIN {X 0,Y 368.924,Z 140.155,A -85,B 0,C 180,E1 -12757.604,E2 -12757.604} C_VEL
LIN {X 0,Y 368.959,Z 140.152,A -85,B 0,C 180,E1 -12761.106,E2 -12761.106} C_VEL
LIN {X 0,Y 368.999,Z 140.141,A -85,B 0,C 180,E1 -12764.535,E2 -12764.535} C_VEL
LIN {X 0,Y 369.006,Z 140.137,A -85,B 0,C 180,E1 -12767.907,E2 -12767.907} C_VEL
LIN {X 0,Y 369.093,Z 140.126,A -85,B 0,C 180,E1 -12771.238,E2 -12771.238} C_VEL
LIN {X 0,Y 369.126,Z 140.13,A -85,B 0,C 180,E1 -12774.537,E2 -12774.537} C_VEL
LIN {X 0,Y 369.315,Z 140.105,A -85,B 0,C 180,E1 -12777.819,E2 -12777.819} C_VEL
LIN {X 0,Y 369.237,Z 140.113,A -85,B 0,C 180,E1 -12781.091,E2 -12781.091} C_VEL
LIN {X 0,Y 369.305,Z 140.109,A -85,B 0,C 180,E1 -12782.181,E2 -12782.181} C_VEL
LIN {X 0,Y 369.162,Z 140.126,A -85,B 0,C 180,E1 -12786.559,E2 -12786.559} C_VEL
LIN {X 0,Y 369.065,Z 140.133,A -85,B 0,C 180,E1 -12789.868,E2 -12789.868} C_VEL
LIN {X 0,Y 369.039,Z 140.135,A -85,B 0,C 180,E1 -12793.772,E2 -12793.772} C_VEL
LIN {X 0,Y 368.979,Z 140.144,A -85,B 0,C 180,E1 -12797.757,E2 -12797.757} C_VEL
LIN {X 0,Y 368.911,Z 140.151,A -85,B 0,C 180,E1 -12801.221,E2 -12801.221} C_VEL
LIN {X 0,Y 368.924,Z 140.148,A -85,B 0,C 180,E1 -12804.778,E2 -12804.778} C_VEL
LIN {X 0,Y 368.894,Z 140.155,A -85,B 0,C 180,E1 -12808.792,E2 -12808.792} C_VEL
LIN {X 0,Y 368.899,Z 140.157,A -85,B 0,C 180,E1 -12812.238,E2 -12812.238} C_VEL
LIN {X 0,Y 368.929,Z 140.15,A -85,B 0,C 180,E1 -12815.001,E2 -12815.001} C_VEL
LIN {X 0,Y 368.877,Z 140.158,A -85,B 0,C 180,E1 -12818.634,E2 -12818.634} C_VEL
LIN {X 0,Y 368.865,Z 140.156,A -85,B 0,C 180,E1 -12822.006,E2 -12822.006} C_VEL
LIN {X 0,Y 368.874,Z 140.161,A -85,B 0,C 180,E1 -12825.175,E2 -12825.175} C_VEL
LIN {X 0,Y 368.865,Z 140.163,A -85,B 0,C 180,E1 -12828.175,E2 -12828.175} C_VEL
LIN {X 0,Y 368.876,Z 140.154,A -85,B 0,C 180,E1 -12831.366,E2 -12831.366} C_VEL
LIN {X 0,Y 368.931,Z 140.152,A -85,B 0,C 180,E1 -12835.146,E2 -12835.146} C_VEL
LIN {X 0,Y 368.935,Z 140.244,A -85,B 0,C 180,E1 -12837.057,E2 -12837.057} C_VEL
LIN {X 0,Y 370.776,Z 147.022,A -85,B 0,C 180,E1 -12838.772,E2 -12838.772} C_VEL
LIN {X 0,Y 380.854,Z 168.137,A -85,B 0,C 180,E1 -12840.147,E2 -12840.147} C_VEL
LIN {X 0,Y 386.736,Z 181.789,A -85,B 0,C 180,E1 -12840.935,E2 -12840.935} C_VEL
LIN {X 0,Y 384.73,Z 266.925,A -85,B 0,C 180,E1 -12842.54,E2 -12842.54} C_VEL
LIN {X 0,Y 383.591,Z 311.511,A -85,B 0,C 180,E1 -12843.402,E2 -12843.402} C_VEL
LIN {X 0,Y 382.865,Z 326.475,A -85,B 0,C 180,E1 -12843.885,E2 -12843.885} C_VEL
LIN {X 0,Y 381.885,Z 340.959,A -85,B 0,C 180,E1 -12844.56,E2 -12844.56} C_VEL
LIN {X 0,Y 380.748,Z 353.431,A -85,B 0,C 180,E1 -12845.315,E2 -12845.315} C_VEL
LIN {X 0,Y 379.22,Z 367.41,A -85,B 0,C 180,E1 -12846.374,E2 -12846.374} C_VEL
LIN {X 0,Y 377.598,Z 380.186,A -85,B 0,C 180,E1 -12847.57,E2 -12847.57} C_VEL
LIN {X 0,Y 375.981,Z 391.988,A -85,B 0,C 180,E1 -12848.91,E2 -12848.91} C_VEL
LIN {X 0,Y 374.581,Z 402.026,A -85,B 0,C 180,E1 -12850.262,E2 -12850.262} C_VEL
LIN {X 0,Y 373.025,Z 412.21,A -85,B 0,C 180,E1 -12851.888,E2 -12851.888} C_VEL
LIN {X 0,Y 371.455,Z 422.174,A -85,B 0,C 180,E1 -12853.795,E2 -12853.795} C_VEL
LIN {X 0,Y 370.169,Z 430.435,A -85,B 0,C 180,E1 -12855.711,E2 -12855.711} C_VEL
LIN {X 0,Y 369.505,Z 436.39,A -85,B 0,C 180,E1 -12857.366,E2 -12857.366} C_VEL
LIN {X 0,Y 368.591,Z 442.946,A -85,B 0,C 180,E1 -12859.564,E2 -12859.564} C_VEL
LIN {X 0,Y 368.055,Z 448.067,A -85,B 0,C 180,E1 -12861.766,E2 -12861.766} C_VEL
LIN {X 0,Y 367.786,Z 451.228,A -85,B 0,C 180,E1 -12863.549,E2 -12863.549} C_VEL
LIN {X 0,Y 367.55,Z 453.906,A -85,B 0,C 180,E1 -12865.613,E2 -12865.613} C_VEL
LIN {X 0,Y 367.442,Z 455.644,A -85,B 0,C 180,E1 -12867.808,E2 -12867.808} C_VEL
LIN {X 0,Y 367.457,Z 456.25,A -85,B 0,C 180,E1 -12870,E2 -12870} C_VEL
LIN {X 0,Y 367.442,Z 455.69,A -85,B 0,C 180,E1 -12872.192,E2 -12872.192} C_VEL
LIN {X 0,Y 367.549,Z 454.013,A -85,B 0,C 180,E1 -12874.387,E2 -12874.387} C_VEL
LIN {X 0,Y 367.798,Z 451.181,A -85,B 0,C 180,E1 -12876.584,E2 -12876.584} C_VEL
LIN {X 0,Y 368.143,Z 447.127,A -85,B 0,C 180,E1 -12878.785,E2 -12878.785} C_VEL
LIN {X 0,Y 368.685,Z 442.139,A -85,B 0,C 180,E1 -12880.84,E2 -12880.84} C_VEL
LIN {X 0,Y 368.31,Z 439.859,A -85,B 0,C 180,E1 -12881.686,E2 -12881.686} C_VEL
LIN {X 0,Y 366.054,Z 435.885,A -85,B 0,C 180,E1 -12883.059,E2 -12883.059} C_VEL
LIN {X 0,Y 363.887,Z 431.511,A -85,B 0,C 180,E1 -12884.414,E2 -12884.414} C_VEL
LIN {X 0,Y 363.658,Z 428.461,A -85,B 0,C 180,E1 -12885.218,E2 -12885.218} C_VEL
LIN {X 0,Y 364.969,Z 420.171,A -85,B 0,C 180,E1 -12887.077,E2 -12887.077} C_VEL
LIN {X 0,Y 366.614,Z 409.759,A -85,B 0,C 180,E1 -12889.02,E2 -12889.02} C_VEL
LIN {X 0,Y 368.289,Z 399.525,A -85,B 0,C 180,E1 -12890.603,E2 -12890.603} C_VEL
LIN {X 0,Y 370.023,Z 387.374,A -85,B 0,C 180,E1 -12892.179,E2 -12892.179} C_VEL
LIN {X 0,Y 371.827,Z 374.608,A -85,B 0,C 180,E1 -12893.534,E2 -12893.534} C_VEL
LIN {X 0,Y 373.419,Z 362.275,A -85,B 0,C 180,E1 -12894.608,E2 -12894.608} C_VEL
LIN {X 0,Y 374.772,Z 349.04,A -85,B 0,C 180,E1 -12895.551,E2 -12895.551} C_VEL
LIN {X 0,Y 376.05,Z 333.604,A -85,B 0,C 180,E1 -12896.394,E2 -12896.394} C_VEL
LIN {X 0,Y 377.034,Z 318.375,A -85,B 0,C 180,E1 -12896.986,E2 -12896.986} C_VEL
LIN {X 0,Y 377.627,Z 303.934,A -85,B 0,C 180,E1 -12897.352,E2 -12897.352} C_VEL
LIN {X 0,Y 380.609,Z 184.45,A -85,B 0,C 180,E1 -12899.633,E2 -12899.633} C_VEL
LIN {X 0,Y 376.974,Z 175.344,A -85,B 0,C 180,E1 -12900.147,E2 -12900.147} C_VEL
LIN {X 0,Y 368.357,Z 156.776,A -85,B 0,C 180,E1 -12901.349,E2 -12901.349} C_VEL
LIN {X 0,Y 363.422,Z 146.898,A -85,B 0,C 180,E1 -12902.074,E2 -12902.074} C_VEL
LIN {X 0,Y 361.862,Z 141.034,A -85,B 0,C 180,E1 -12903.679,E2 -12903.679} C_VEL
LIN {X 0,Y 361.857,Z 141.035,A -85,B 0,C 180,E1 -12907.221,E2 -12907.221} C_VEL
LIN {X 0,Y 361.811,Z 141.039,A -85,B 0,C 180,E1 -12910.751,E2 -12910.751} C_VEL
LIN {X 0,Y 361.812,Z 141.04,A -85,B 0,C 180,E1 -12914.37,E2 -12914.37} C_VEL
LIN {X 0,Y 361.823,Z 141.024,A -85,B 0,C 180,E1 -12917.571,E2 -12917.571} C_VEL
LIN {X 0,Y 361.843,Z 141.028,A -85,B 0,C 180,E1 -12921.572,E2 -12921.572} C_VEL
LIN {X 0,Y 361.871,Z 141.03,A -85,B 0,C 180,E1 -12924.656,E2 -12924.656} C_VEL
LIN {X 0,Y 361.848,Z 141.027,A -85,B 0,C 180,E1 -12927.055,E2 -12927.055} C_VEL
LIN {X 0,Y 361.868,Z 141.031,A -85,B 0,C 180,E1 -12930.952,E2 -12930.952} C_VEL
LIN {X 0,Y 361.862,Z 141.033,A -85,B 0,C 180,E1 -12934.705,E2 -12934.705} C_VEL
LIN {X 0,Y 361.856,Z 141.031,A -85,B 0,C 180,E1 -12938.345,E2 -12938.345} C_VEL
LIN {X 0,Y 361.906,Z 141.023,A -85,B 0,C 180,E1 -12942.093,E2 -12942.093} C_VEL
LIN {X 0,Y 361.997,Z 141.011,A -85,B 0,C 180,E1 -12946.103,E2 -12946.103} C_VEL
LIN {X 0,Y 362.002,Z 141.012,A -85,B 0,C 180,E1 -12949.937,E2 -12949.937} C_VEL
LIN {X 0,Y 362.122,Z 141.002,A -85,B 0,C 180,E1 -12953.313,E2 -12953.313} C_VEL
LIN {X 0,Y 362.267,Z 140.987,A -85,B 0,C 180,E1 -12957.776,E2 -12957.776} C_VEL
LIN {X 0,Y 362.179,Z 140.989,A -85,B 0,C 180,E1 -12961.112,E2 -12961.112} C_VEL
LIN {X 0,Y 362.279,Z 140.982,A -85,B 0,C 180,E1 -12962.223,E2 -12962.223} C_VEL
LIN {X 0,Y 362.127,Z 141,A -85,B 0,C 180,E1 -12966.687,E2 -12966.687} C_VEL
LIN {X 0,Y 362.003,Z 141.015,A -85,B 0,C 180,E1 -12970.063,E2 -12970.063} C_VEL
